LIN {X 0,Y 523.894,Z 140.721,A -85,B 0,C 180,E1 -4799.759,E2 -4799.759} C_VEL
LIN {X 0,Y 523.931,Z 140.719,A -85,B 0,C 180,E1 -4802.45,E2 -4802.45} C_VEL
LIN {X 0,Y 523.92,Z 140.722,A -85,B 0,C 180,E1 -4805.227,E2 -4805.227} C_VEL
LIN {X 0,Y 523.914,Z 140.72,A -85,B 0,C 180,E1 -4808.102,E2 -4808.102} C_VEL
LIN {X 0,Y 523.94,Z 140.717,A -85,B 0,C 180,E1 -4811.308,E2 -4811.308} C_VEL
LIN {X 0,Y 523.938,Z 140.723,A -85,B 0,C 180,E1 -4814.689,E2 -4814.689} C_VEL
LIN {X 0,Y 523.94,Z 140.717,A -85,B 0,C 180,E1 -4817.88,E2 -4817.88} C_VEL
LIN {X 0,Y 523.92,Z 140.72,A -85,B 0,C 180,E1 -4820.915,E2 -4820.915} C_VEL
LIN {X 0,Y 523.895,Z 140.724,A -85,B 0,C 180,E1 -4823.825,E2 -4823.825} C_VEL
LIN {X 0,Y 523.941,Z 140.719,A -85,B 0,C 180,E1 -4826.635,E2 -4826.635} C_VEL
LIN {X 0,Y 523.947,Z 140.715,A -85,B 0,C 180,E1 -4829.355,E2 -4829.355} C_VEL
LIN {X 0,Y 523.946,Z 140.721,A -85,B 0,C 180,E1 -4832.288,E2 -4832.288} C_VEL
LIN {X 0,Y 523.927,Z 140.719,A -85,B 0,C 180,E1 -4834.58,E2 -4834.58} C_VEL
LIN {X 0,Y 523.91,Z 140.72,A -85,B 0,C 180,E1 -4837.106,E2 -4837.106} C_VEL
LIN {X 0,Y 523.978,Z 140.72,A -85,B 0,C 180,E1 -4839.866,E2 -4839.866} C_VEL
LIN {X 0,Y 523.953,Z 140.714,A -85,B 0,C 180,E1 -4842.837,E2 -4842.837} C_VEL
LIN {X 0,Y 523.977,Z 140.714,A -85,B 0,C 180,E1 -4845.236,E2 -4845.236} C_VEL
LIN {X 0,Y 524.012,Z 140.707,A -85,B 0,C 180,E1 -4848.394,E2 -4848.394} C_VEL
LIN {X 0,Y 524,Z 140.717,A -85,B 0,C 180,E1 -4851.516,E2 -4851.516} C_VEL
LIN {X 0,Y 524.082,Z 140.699,A -85,B 0,C 180,E1 -4854.614,E2 -4854.614} C_VEL
LIN {X 0,Y 524.113,Z 140.698,A -85,B 0,C 180,E1 -4857.695,E2 -4857.695} C_VEL
LIN {X 0,Y 524.121,Z 140.696,A -85,B 0,C 180,E1 -4860.768,E2 -4860.768} C_VEL
LIN {X 0,Y 524.071,Z 140.708,A -85,B 0,C 180,E1 -4863.075,E2 -4863.075} C_VEL
LIN {X 0,Y 524.034,Z 140.704,A -85,B 0,C 180,E1 -4866.159,E2 -4866.159} C_VEL
LIN {X 0,Y 524.001,Z 140.711,A -85,B 0,C 180,E1 -4868.484,E2 -4868.484} C_VEL
LIN {X 0,Y 524.003,Z 140.708,A -85,B 0,C 180,E1 -4871.74,E2 -4871.74} C_VEL
LIN {X 0,Y 523.993,Z 140.714,A -85,B 0,C 180,E1 -4875.052,E2 -4875.052} C_VEL
LIN {X 0,Y 523.964,Z 140.713,A -85,B 0,C 180,E1 -4877.969,E2 -4877.969} C_VEL
LIN {X 0,Y 523.972,Z 140.717,A -85,B 0,C 180,E1 -4880.41,E2 -4880.41} C_VEL
LIN {X 0,Y 523.911,Z 140.723,A -85,B 0,C 180,E1 -4882.894,E2 -4882.894} C_VEL
LIN {X 0,Y 523.953,Z 140.714,A -85,B 0,C 180,E1 -4885.419,E2 -4885.419} C_VEL
LIN {X 0,Y 523.968,Z 140.716,A -85,B 0,C 180,E1 -4887.999,E2 -4887.999} C_VEL
LIN {X 0,Y 523.945,Z 140.717,A -85,B 0,C 180,E1 -4890.855,E2 -4890.855} C_VEL
LIN {X 0,Y 523.96,Z 140.716,A -85,B 0,C 180,E1 -4893.735,E2 -4893.735} C_VEL
LIN {X 0,Y 523.904,Z 140.725,A -85,B 0,C 180,E1 -4896.402,E2 -4896.402} C_VEL
LIN {X 0,Y 523.924,Z 140.718,A -85,B 0,C 180,E1 -4899.085,E2 -4899.085} C_VEL
LIN {X 0,Y 523.957,Z 140.72,A -85,B 0,C 180,E1 -4902.119,E2 -4902.119} C_VEL
LIN {X 0,Y 523.957,Z 140.715,A -85,B 0,C 180,E1 -4905.309,E2 -4905.309} C_VEL
LIN {X 0,Y 523.921,Z 140.718,A -85,B 0,C 180,E1 -4906.898,E2 -4906.898} C_VEL
LIN {X 0,Y 523.254,Z 140.808,A -85,B 0,C 180,E1 -4907.54,E2 -4907.54} C_VEL
LIN {X 0,Y 520.412,Z 141.161,A -85,B 0,C 180,E1 -4908.581,E2 -4908.581} C_VEL
LIN {X 0,Y 518.008,Z 141.461,A -85,B 0,C 180,E1 -4909.42,E2 -4909.42} C_VEL
LIN {X 0,Y 516.971,Z 141.589,A -85,B 0,C 180,E1 -4910.068,E2 -4910.068} C_VEL
LIN {X 0,Y 516.883,Z 141.597,A -85,B 0,C 180,E1 -4910.287,E2 -4910.287} C_VEL
LIN {X 0,Y 516.879,Z 141.6,A -85,B 0,C 180,E1 -4913.343,E2 -4913.343} C_VEL
LIN {X 0,Y 516.886,Z 141.596,A -85,B 0,C 180,E1 -4916.119,E2 -4916.119} C_VEL
LIN {X 0,Y 516.892,Z 141.596,A -85,B 0,C 180,E1 -4918.936,E2 -4918.936} C_VEL
LIN {X 0,Y 516.918,Z 141.598,A -85,B 0,C 180,E1 -4921.585,E2 -4921.585} C_VEL
LIN {X 0,Y 516.934,Z 141.59,A -85,B 0,C 180,E1 -4924.211,E2 -4924.211} C_VEL
LIN {X 0,Y 516.867,Z 141.601,A -85,B 0,C 180,E1 -4926.776,E2 -4926.776} C_VEL
LIN {X 0,Y 516.972,Z 141.775,A -85,B 0,C 180,E1 -4929.041,E2 -4929.041} C_VEL
LIN {X 0,Y 517.715,Z 147.463,A -85,B 0,C 180,E1 -4930.161,E2 -4930.161} C_VEL
LIN {X 0,Y 517.441,Z 161.62,A -85,B 0,C 180,E1 -4932.818,E2 -4932.818} C_VEL
LIN {X 0,Y 517.249,Z 171.826,A -85,B 0,C 180,E1 -4934.685,E2 -4934.685} C_VEL
LIN {X 0,Y 519.153,Z 182.577,A -85,B 0,C 180,E1 -4934.898,E2 -4934.898} C_VEL
LIN {X 0,Y 518.664,Z 279.186,A -85,B 0,C 180,E1 -4936.258,E2 -4936.258} C_VEL
LIN {X 0,Y 518.488,Z 292.359,A -85,B 0,C 180,E1 -4936.603,E2 -4936.603} C_VEL
LIN {X 0,Y 518.232,Z 304.457,A -85,B 0,C 180,E1 -4937.07,E2 -4937.07} C_VEL
LIN {X 0,Y 518.017,Z 315.553,A -85,B 0,C 180,E1 -4937.644,E2 -4937.644} C_VEL
LIN {X 0,Y 517.72,Z 326.26,A -85,B 0,C 180,E1 -4938.35,E2 -4938.35} C_VEL
LIN {X 0,Y 517.414,Z 336.963,A -85,B 0,C 180,E1 -4939.236,E2 -4939.236} C_VEL
LIN {X 0,Y 517.104,Z 346.594,A -85,B 0,C 180,E1 -4940.219,E2 -4940.219} C_VEL
LIN {X 0,Y 516.877,Z 354.481,A -85,B 0,C 180,E1 -4941.201,E2 -4941.201} C_VEL
LIN {X 0,Y 516.638,Z 362.196,A -85,B 0,C 180,E1 -4942.378,E2 -4942.378} C_VEL
LIN {X 0,Y 516.501,Z 369.27,A -85,B 0,C 180,E1 -4943.751,E2 -4943.751} C_VEL
LIN {X 0,Y 516.316,Z 373.987,A -85,B 0,C 180,E1 -4944.924,E2 -4944.924} C_VEL
LIN {X 0,Y 516.375,Z 377.597,A -85,B 0,C 180,E1 -4946.098,E2 -4946.098} C_VEL
LIN {X 0,Y 516.327,Z 379.464,A -85,B 0,C 180,E1 -4946.879,E2 -4946.879} C_VEL
LIN {X 0,Y 516.266,Z 380.874,A -85,B 0,C 180,E1 -4947.659,E2 -4947.659} C_VEL
LIN {X 0,Y 516.163,Z 382.495,A -85,B 0,C 180,E1 -4949.22,E2 -4949.22} C_VEL
LIN {X 0,Y 516.158,Z 382.733,A -85,B 0,C 180,E1 -4950,E2 -4950} C_VEL
LIN {X 0,Y 516.163,Z 382.55,A -85,B 0,C 180,E1 -4950.78,E2 -4950.78} C_VEL
LIN {X 0,Y 516.266,Z 381,A -85,B 0,C 180,E1 -4952.341,E2 -4952.341} C_VEL
LIN {X 0,Y 516.327,Z 379.645,A -85,B 0,C 180,E1 -4953.121,E2 -4953.121} C_VEL
LIN {X 0,Y 516.368,Z 376.78,A -85,B 0,C 180,E1 -4954.293,E2 -4954.293} C_VEL
LIN {X 0,Y 516.408,Z 372.896,A -85,B 0,C 180,E1 -4955.467,E2 -4955.467} C_VEL
LIN {X 0,Y 516.504,Z 366.966,A -85,B 0,C 180,E1 -4956.828,E2 -4956.828} C_VEL
LIN {X 0,Y 516.681,Z 360.354,A -85,B 0,C 180,E1 -4958.014,E2 -4958.014} C_VEL
LIN {X 0,Y 516.904,Z 352.199,A -85,B 0,C 180,E1 -4959.193,E2 -4959.193} C_VEL
LIN {X 0,Y 517.155,Z 343.853,A -85,B 0,C 180,E1 -4960.176,E2 -4960.176} C_VEL
LIN {X 0,Y 517.485,Z 333.549,A -85,B 0,C 180,E1 -4961.159,E2 -4961.159} C_VEL
LIN {X 0,Y 517.828,Z 322.274,A -85,B 0,C 180,E1 -4962.02,E2 -4962.02} C_VEL
LIN {X 0,Y 518.131,Z 310.364,A -85,B 0,C 180,E1 -4962.733,E2 -4962.733} C_VEL
LIN {X 0,Y 518.385,Z 298.344,A -85,B 0,C 180,E1 -4963.275,E2 -4963.275} C_VEL
LIN {X 0,Y 518.593,Z 285.267,A -85,B 0,C 180,E1 -4963.694,E2 -4963.694} C_VEL
LIN {X 0,Y 518.78,Z 272.765,A -85,B 0,C 180,E1 -4963.939,E2 -4963.939} C_VEL
LIN {X 0,Y 519.06,Z 182.069,A -85,B 0,C 180,E1 -4965.202,E2 -4965.202} C_VEL
LIN {X 0,Y 517.238,Z 171.844,A -85,B 0,C 180,E1 -4965.403,E2 -4965.403} C_VEL
LIN {X 0,Y 517.612,Z 155.547,A -85,B 0,C 180,E1 -4968.402,E2 -4968.402} C_VEL
LIN {X 0,Y 517.682,Z 146.406,A -85,B 0,C 180,E1 -4970.132,E2 -4970.132} C_VEL
LIN {X 0,Y 516.95,Z 141.595,A -85,B 0,C 180,E1 -4971.117,E2 -4971.117} C_VEL
LIN {X 0,Y 516.898,Z 141.598,A -85,B 0,C 180,E1 -4974.36,E2 -4974.36} C_VEL
LIN {X 0,Y 516.926,Z 141.598,A -85,B 0,C 180,E1 -4976.658,E2 -4976.658} C_VEL
LIN {X 0,Y 516.911,Z 141.592,A -85,B 0,C 180,E1 -4979.523,E2 -4979.523} C_VEL
LIN {X 0,Y 516.896,Z 141.602,A -85,B 0,C 180,E1 -4982.543,E2 -4982.543} C_VEL
LIN {X 0,Y 516.867,Z 141.597,A -85,B 0,C 180,E1 -4985.329,E2 -4985.329} C_VEL
LIN {X 0,Y 516.882,Z 141.598,A -85,B 0,C 180,E1 -4987.943,E2 -4987.943} C_VEL
LIN {X 0,Y 516.884,Z 141.598,A -85,B 0,C 180,E1 -4990.741,E2 -4990.741} C_VEL
LIN {X 0,Y 516.885,Z 141.596,A -85,B 0,C 180,E1 -4992.831,E2 -4992.831} C_VEL
LIN {X 0,Y 516.924,Z 141.59,A -85,B 0,C 180,E1 -4995.01,E2 -4995.01} C_VEL
LIN {X 0,Y 516.915,Z 141.595,A -85,B 0,C 180,E1 -4998.398,E2 -4998.398} C_VEL
LIN {X 0,Y 516.883,Z 141.596,A -85,B 0,C 180,E1 -5001.284,E2 -5001.284} C_VEL
LIN {X 0,Y 516.871,Z 141.601,A -85,B 0,C 180,E1 -5004.219,E2 -5004.219} C_VEL
LIN {X 0,Y 516.895,Z 141.594,A -85,B 0,C 180,E1 -5007.053,E2 -5007.053} C_VEL
LIN {X 0,Y 516.892,Z 141.602,A -85,B 0,C 180,E1 -5009.796,E2 -5009.796} C_VEL
LIN {X 0,Y 516.926,Z 141.59,A -85,B 0,C 180,E1 -5012.467,E2 -5012.467} C_VEL
LIN {X 0,Y 516.909,Z 141.594,A -85,B 0,C 180,E1 -5015.072,E2 -5015.072} C_VEL
LIN {X 0,Y 516.885,Z 141.595,A -85,B 0,C 180,E1 -5018.462,E2 -5018.462} C_VEL
LIN {X 0,Y 516.903,Z 141.595,A -85,B 0,C 180,E1 -5020.955,E2 -5020.955} C_VEL
LIN {X 0,Y 516.913,Z 141.599,A -85,B 0,C 180,E1 -5023.41,E2 -5023.41} C_VEL
LIN {X 0,Y 516.894,Z 141.595,A -85,B 0,C 180,E1 -5025.834,E2 -5025.834} C_VEL
LIN {X 0,Y 516.965,Z 141.585,A -85,B 0,C 180,E1 -5028.234,E2 -5028.234} C_VEL
LIN {X 0,Y 516.968,Z 141.589,A -85,B 0,C 180,E1 -5031.4,E2 -5031.4} C_VEL
LIN {X 0,Y 517.002,Z 141.581,A -85,B 0,C 180,E1 -5033.757,E2 -5033.757} C_VEL
LIN {X 0,Y 517.012,Z 141.588,A -85,B 0,C 180,E1 -5036.883,E2 -5036.883} C_VEL
LIN {X 0,Y 517.085,Z 141.57,A -85,B 0,C 180,E1 -5040,E2 -5040} C_VEL
LIN {X 0,Y 517.01,Z 141.582,A -85,B 0,C 180,E1 -5043.117,E2 -5043.117} C_VEL
LIN {X 0,Y 517.002,Z 141.584,A -85,B 0,C 180,E1 -5046.243,E2 -5046.243} C_VEL
LIN {X 0,Y 516.944,Z 141.587,A -85,B 0,C 180,E1 -5049.389,E2 -5049.389} C_VEL
LIN {X 0,Y 516.951,Z 141.587,A -85,B 0,C 180,E1 -5051.807,E2 -5051.807} C_VEL
LIN {X 0,Y 516.944,Z 141.588,A -85,B 0,C 180,E1 -5055.147,E2 -5055.147} C_VEL
LIN {X 0,Y 516.915,Z 141.599,A -85,B 0,C 180,E1 -5058.223,E2 -5058.223} C_VEL
LIN {X 0,Y 516.911,Z 141.593,A -85,B 0,C 180,E1 -5060.702,E2 -5060.702} C_VEL
LIN {X 0,Y 516.889,Z 141.603,A -85,B 0,C 180,E1 -5064.073,E2 -5064.073} C_VEL
LIN {X 0,Y 516.92,Z 141.591,A -85,B 0,C 180,E1 -5066.658,E2 -5066.658} C_VEL
LIN {X 0,Y 516.909,Z 141.595,A -85,B 0,C 180,E1 -5069.524,E2 -5069.524} C_VEL
LIN {X 0,Y 516.895,Z 141.594,A -85,B 0,C 180,E1 -5072.543,E2 -5072.543} C_VEL
LIN {X 0,Y 516.863,Z 141.601,A -85,B 0,C 180,E1 -5075.329,E2 -5075.329} C_VEL
LIN {X 0,Y 516.878,Z 141.6,A -85,B 0,C 180,E1 -5077.943,E2 -5077.943} C_VEL
LIN {X 0,Y 516.88,Z 141.595,A -85,B 0,C 180,E1 -5080.742,E2 -5080.742} C_VEL
LIN {X 0,Y 516.881,Z 141.598,A -85,B 0,C 180,E1 -5083.904,E2 -5083.904} C_VEL
LIN {X 0,Y 516.88,Z 141.596,A -85,B 0,C 180,E1 -5086.107,E2 -5086.107} C_VEL
LIN {X 0,Y 516.902,Z 141.593,A -85,B 0,C 180,E1 -5088.4,E2 -5088.4} C_VEL
LIN {X 0,Y 516.877,Z 141.604,A -85,B 0,C 180,E1 -5091.284,E2 -5091.284} C_VEL
LIN {X 0,Y 516.871,Z 141.596,A -85,B 0,C 180,E1 -5094.22,E2 -5094.22} C_VEL
LIN {X 0,Y 516.88,Z 141.604,A -85,B 0,C 180,E1 -5097.052,E2 -5097.052} C_VEL
LIN {X 0,Y 516.863,Z 141.6,A -85,B 0,C 180,E1 -5099.795,E2 -5099.795} C_VEL
LIN {X 0,Y 516.877,Z 141.599,A -85,B 0,C 180,E1 -5102.465,E2 -5102.465} C_VEL
LIN {X 0,Y 516.846,Z 141.608,A -85,B 0,C 180,E1 -5105.069,E2 -5105.069} C_VEL
LIN {X 0,Y 516.902,Z 141.692,A -85,B 0,C 180,E1 -5105.981,E2 -5105.981} C_VEL
LIN {X 0,Y 518.288,Z 149.569,A -85,B 0,C 180,E1 -5107.372,E2 -5107.372} C_VEL
LIN {X 0,Y 517.935,Z 164.192,A -85,B 0,C 180,E1 -5109.793,E2 -5109.793} C_VEL
LIN {X 0,Y 517.529,Z 180.375,A -85,B 0,C 180,E1 -5112.437,E2 -5112.437} C_VEL
LIN {X 0,Y 517.238,Z 194.025,A -85,B 0,C 180,E1 -5114.635,E2 -5114.635} C_VEL
LIN {X 0,Y 519.105,Z 206.824,A -85,B 0,C 180,E1 -5114.871,E2 -5114.871} C_VEL
LIN {X 0,Y 518.632,Z 301.977,A -85,B 0,C 180,E1 -5116.207,E2 -5116.207} C_VEL
LIN {X 0,Y 518.385,Z 315.258,A -85,B 0,C 180,E1 -5116.55,E2 -5116.55} C_VEL
LIN {X 0,Y 518.1,Z 328.548,A -85,B 0,C 180,E1 -5117.067,E2 -5117.067} C_VEL
LIN {X 0,Y 517.775,Z 340.338,A -85,B 0,C 180,E1 -5117.696,E2 -5117.696} C_VEL
LIN {X 0,Y 517.491,Z 352.593,A -85,B 0,C 180,E1 -5118.544,E2 -5118.544} C_VEL
LIN {X 0,Y 517.171,Z 362.784,A -85,B 0,C 180,E1 -5119.429,E2 -5119.429} C_VEL
LIN {X 0,Y 516.926,Z 371.954,A -85,B 0,C 180,E1 -5120.413,E2 -5120.413} C_VEL
LIN {X 0,Y 516.653,Z 380.888,A -85,B 0,C 180,E1 -5121.591,E2 -5121.591} C_VEL
LIN {X 0,Y 516.503,Z 388.079,A -85,B 0,C 180,E1 -5122.769,E2 -5122.769} C_VEL
LIN {X 0,Y 516.407,Z 394.627,A -85,B 0,C 180,E1 -5124.142,E2 -5124.142} C_VEL
LIN {X 0,Y 516.267,Z 398.957,A -85,B 0,C 180,E1 -5125.315,E2 -5125.315} C_VEL
LIN {X 0,Y 516.352,Z 401.252,A -85,B 0,C 180,E1 -5126.098,E2 -5126.098} C_VEL
LIN {X 0,Y 516.282,Z 403.109,A -85,B 0,C 180,E1 -5126.879,E2 -5126.879} C_VEL
LIN {X 0,Y 516.261,Z 404.502,A -85,B 0,C 180,E1 -5127.659,E2 -5127.659} C_VEL
LIN {X 0,Y 516.161,Z 406.101,A -85,B 0,C 180,E1 -5129.22,E2 -5129.22} C_VEL
LIN {X 0,Y 516.157,Z 406.317,A -85,B 0,C 180,E1 -5130,E2 -5130} C_VEL
LIN {X 0,Y 516.192,Z 405.496,A -85,B 0,C 180,E1 -5131.56,E2 -5131.56} C_VEL
LIN {X 0,Y 516.261,Z 404.505,A -85,B 0,C 180,E1 -5132.341,E2 -5132.341} C_VEL
LIN {X 0,Y 516.282,Z 403.112,A -85,B 0,C 180,E1 -5133.121,E2 -5133.121} C_VEL
LIN {X 0,Y 516.31,Z 400.182,A -85,B 0,C 180,E1 -5134.294,E2 -5134.294} C_VEL
LIN {X 0,Y 516.39,Z 396.216,A -85,B 0,C 180,E1 -5135.467,E2 -5135.467} C_VEL
LIN {X 0,Y 516.442,Z 390.346,A -85,B 0,C 180,E1 -5136.794,E2 -5136.794} C_VEL
LIN {X 0,Y 516.587,Z 383.445,A -85,B 0,C 180,E1 -5138.016,E2 -5138.016} C_VEL
LIN {X 0,Y 516.806,Z 375.171,A -85,B 0,C 180,E1 -5139.195,E2 -5139.195} C_VEL
LIN {X 0,Y 517.021,Z 366.689,A -85,B 0,C 180,E1 -5140.178,E2 -5140.178} C_VEL
LIN {X 0,Y 517.372,Z 356.209,A -85,B 0,C 180,E1 -5141.161,E2 -5141.161} C_VEL
LIN {X 0,Y 517.674,Z 345.063,A -85,B 0,C 180,E1 -5142.003,E2 -5142.003} C_VEL
LIN {X 0,Y 517.96,Z 334.472,A -85,B 0,C 180,E1 -5142.638,E2 -5142.638} C_VEL
LIN {X 0,Y 518.236,Z 322.813,A -85,B 0,C 180,E1 -5143.179,E2 -5143.179} C_VEL
LIN {X 0,Y 518.494,Z 309.377,A -85,B 0,C 180,E1 -5143.622,E2 -5143.622} C_VEL
LIN {X 0,Y 518.708,Z 296.109,A -85,B 0,C 180,E1 -5143.891,E2 -5143.891} C_VEL
LIN {X 0,Y 518.988,Z 204.886,A -85,B 0,C 180,E1 -5145.16,E2 -5145.16} C_VEL
LIN {X 0,Y 517.226,Z 193.828,A -85,B 0,C 180,E1 -5145.388,E2 -5145.388} C_VEL
LIN {X 0,Y 517.68,Z 175.231,A -85,B 0,C 180,E1 -5148.399,E2 -5148.399} C_VEL
LIN {X 0,Y 518.165,Z 157.709,A -85,B 0,C 180,E1 -5151.273,E2 -5151.273} C_VEL
LIN {X 0,Y 518.259,Z 148.792,A -85,B 0,C 180,E1 -5152.759,E2 -5152.759} C_VEL
LIN {X 0,Y 516.887,Z 141.601,A -85,B 0,C 180,E1 -5154.073,E2 -5154.073} C_VEL
LIN {X 0,Y 516.85,Z 141.604,A -85,B 0,C 180,E1 -5156.662,E2 -5156.662} C_VEL
LIN {X 0,Y 516.886,Z 141.596,A -85,B 0,C 180,E1 -5159.518,E2 -5159.518} C_VEL
LIN {X 0,Y 516.892,Z 141.597,A -85,B 0,C 180,E1 -5162.542,E2 -5162.542} C_VEL
LIN {X 0,Y 516.866,Z 141.6,A -85,B 0,C 180,E1 -5165.329,E2 -5165.329} C_VEL
LIN {X 0,Y 516.879,Z 141.596,A -85,B 0,C 180,E1 -5167.943,E2 -5167.943} C_VEL
LIN {X 0,Y 516.864,Z 141.606,A -85,B 0,C 180,E1 -5170.743,E2 -5170.743} C_VEL
LIN {X 0,Y 516.854,Z 141.604,A -85,B 0,C 180,E1 -5172.834,E2 -5172.834} C_VEL
LIN {X 0,Y 516.895,Z 141.596,A -85,B 0,C 180,E1 -5175.007,E2 -5175.007} C_VEL
LIN {X 0,Y 516.908,Z 141.6,A -85,B 0,C 180,E1 -5178.399,E2 -5178.399} C_VEL
LIN {X 0,Y 516.88,Z 141.595,A -85,B 0,C 180,E1 -5181.284,E2 -5181.284} C_VEL
LIN {X 0,Y 516.867,Z 141.605,A -85,B 0,C 180,E1 -5184.219,E2 -5184.219} C_VEL
LIN {X 0,Y 516.894,Z 141.594,A -85,B 0,C 180,E1 -5187.053,E2 -5187.053} C_VEL
LIN {X 0,Y 516.885,Z 141.599,A -85,B 0,C 180,E1 -5189.796,E2 -5189.796} C_VEL
LIN {X 0,Y 516.898,Z 141.596,A -85,B 0,C 180,E1 -5192.466,E2 -5192.466} C_VEL
LIN {X 0,Y 516.865,Z 141.597,A -85,B 0,C 180,E1 -5195.069,E2 -5195.069} C_VEL
LIN {X 0,Y 516.868,Z 141.602,A -85,B 0,C 180,E1 -5197.621,E2 -5197.621} C_VEL
LIN {X 0,Y 516.931,Z 141.593,A -85,B 0,C 180,E1 -5200.13,E2 -5200.13} C_VEL
LIN {X 0,Y 516.905,Z 141.592,A -85,B 0,C 180,E1 -5202.595,E2 -5202.595} C_VEL
LIN {X 0,Y 516.942,Z 141.589,A -85,B 0,C 180,E1 -5205.03,E2 -5205.03} C_VEL
LIN {X 0,Y 516.965,Z 141.586,A -85,B 0,C 180,E1 -5208.234,E2 -5208.234} C_VEL
LIN {X 0,Y 516.965,Z 141.592,A -85,B 0,C 180,E1 -5211.4,E2 -5211.4} C_VEL
LIN {X 0,Y 517.002,Z 141.584,A -85,B 0,C 180,E1 -5213.757,E2 -5213.757} C_VEL
LIN {X 0,Y 517.01,Z 141.582,A -85,B 0,C 180,E1 -5216.883,E2 -5216.883} C_VEL
LIN {X 0,Y 517.085,Z 141.57,A -85,B 0,C 180,E1 -5220,E2 -5220} C_VEL
LIN {X 0,Y 517.012,Z 141.588,A -85,B 0,C 180,E1 -5223.117,E2 -5223.117} C_VEL
LIN {X 0,Y 516.995,Z 141.581,A -85,B 0,C 180,E1 -5226.243,E2 -5226.243} C_VEL
LIN {X 0,Y 516.965,Z 141.588,A -85,B 0,C 180,E1 -5228.6,E2 -5228.6} C_VEL
LIN {X 0,Y 516.952,Z 141.586,A -85,B 0,C 180,E1 -5231.807,E2 -5231.807} C_VEL
LIN {X 0,Y 516.944,Z 141.591,A -85,B 0,C 180,E1 -5235.147,E2 -5235.147} C_VEL
LIN {X 0,Y 516.925,Z 141.592,A -85,B 0,C 180,E1 -5238.222,E2 -5238.222} C_VEL
LIN {X 0,Y 516.913,Z 141.599,A -85,B 0,C 180,E1 -5240.702,E2 -5240.702} C_VEL
LIN {X 0,Y 516.904,Z 141.595,A -85,B 0,C 180,E1 -5244.073,E2 -5244.073} C_VEL
LIN {X 0,Y 516.925,Z 141.595,A -85,B 0,C 180,E1 -5246.658,E2 -5246.658} C_VEL
LIN {X 0,Y 516.911,Z 141.592,A -85,B 0,C 180,E1 -5249.524,E2 -5249.524} C_VEL
LIN {X 0,Y 516.896,Z 141.598,A -85,B 0,C 180,E1 -5252.544,E2 -5252.544} C_VEL
LIN {X 0,Y 516.867,Z 141.597,A -85,B 0,C 180,E1 -5255.33,E2 -5255.33} C_VEL
LIN {X 0,Y 516.882,Z 141.602,A -85,B 0,C 180,E1 -5257.943,E2 -5257.943} C_VEL
LIN {X 0,Y 516.886,Z 141.595,A -85,B 0,C 180,E1 -5260.742,E2 -5260.742} C_VEL
LIN {X 0,Y 516.885,Z 141.595,A -85,B 0,C 180,E1 -5262.831,E2 -5262.831} C_VEL
LIN {X 0,Y 516.924,Z 141.59,A -85,B 0,C 180,E1 -5265.01,E2 -5265.01} C_VEL
LIN {X 0,Y 516.917,Z 141.592,A -85,B 0,C 180,E1 -5268.399,E2 -5268.399} C_VEL
LIN {X 0,Y 516.883,Z 141.597,A -85,B 0,C 180,E1 -5270.287,E2 -5270.287} C_VEL
LIN {X 0,Y 516.211,Z 141.679,A -85,B 0,C 180,E1 -5270.937,E2 -5270.937} C_VEL
LIN {X 0,Y 513.365,Z 142.042,A -85,B 0,C 180,E1 -5271.993,E2 -5271.993} C_VEL
LIN {X 0,Y 510.957,Z 142.347,A -85,B 0,C 180,E1 -5272.843,E2 -5272.843} C_VEL
LIN {X 0,Y 509.913,Z 142.474,A -85,B 0,C 180,E1 -5273.499,E2 -5273.499} C_VEL
LIN {X 0,Y 509.822,Z 142.482,A -85,B 0,C 180,E1 -5273.722,E2 -5273.722} C_VEL
LIN {X 0,Y 509.843,Z 142.472,A -85,B 0,C 180,E1 -5276.538,E2 -5276.538} C_VEL
LIN {X 0,Y 509.845,Z 142.479,A -85,B 0,C 180,E1 -5279.334,E2 -5279.334} C_VEL
LIN {X 0,Y 509.892,Z 142.467,A -85,B 0,C 180,E1 -5282.055,E2 -5282.055} C_VEL
LIN {X 0,Y 509.878,Z 142.471,A -85,B 0,C 180,E1 -5284.704,E2 -5284.704} C_VEL
LIN {X 0,Y 509.829,Z 142.48,A -85,B 0,C 180,E1 -5287.458,E2 -5287.458} C_VEL
LIN {X 0,Y 509.909,Z 142.617,A -85,B 0,C 180,E1 -5288.895,E2 -5288.895} C_VEL
LIN {X 0,Y 510.762,Z 148.591,A -85,B 0,C 180,E1 -5290.089,E2 -5290.089} C_VEL
LIN {X 0,Y 510.48,Z 161.707,A -85,B 0,C 180,E1 -5292.576,E2 -5292.576} C_VEL
LIN {X 0,Y 510.268,Z 171.957,A -85,B 0,C 180,E1 -5294.47,E2 -5294.47} C_VEL
LIN {X 0,Y 512.319,Z 183.37,A -85,B 0,C 180,E1 -5294.7,E2 -5294.7} C_VEL
LIN {X 0,Y 511.789,Z 279.376,A -85,B 0,C 180,E1 -5296.07,E2 -5296.07} C_VEL
LIN {X 0,Y 511.585,Z 292.541,A -85,B 0,C 180,E1 -5296.418,E2 -5296.418} C_VEL
LIN {X 0,Y 511.29,Z 305.746,A -85,B 0,C 180,E1 -5296.942,E2 -5296.942} C_VEL
LIN {X 0,Y 510.991,Z 318.287,A -85,B 0,C 180,E1 -5297.633,E2 -5297.633} C_VEL
LIN {X 0,Y 510.709,Z 329.005,A -85,B 0,C 180,E1 -5298.389,E2 -5298.389} C_VEL
LIN {X 0,Y 510.357,Z 339.261,A -85,B 0,C 180,E1 -5299.286,E2 -5299.286} C_VEL
LIN {X 0,Y 510.062,Z 348.463,A -85,B 0,C 180,E1 -5300.283,E2 -5300.283} C_VEL
LIN {X 0,Y 509.747,Z 357.393,A -85,B 0,C 180,E1 -5301.477,E2 -5301.477} C_VEL
LIN {X 0,Y 509.517,Z 364.584,A -85,B 0,C 180,E1 -5302.67,E2 -5302.67} C_VEL
LIN {X 0,Y 509.429,Z 369.435,A -85,B 0,C 180,E1 -5303.664,E2 -5303.664} C_VEL
LIN {X 0,Y 509.251,Z 374.152,A -85,B 0,C 180,E1 -5304.853,E2 -5304.853} C_VEL
LIN {X 0,Y 509.307,Z 377.76,A -85,B 0,C 180,E1 -5306.044,E2 -5306.044} C_VEL
LIN {X 0,Y 509.241,Z 379.628,A -85,B 0,C 180,E1 -5306.835,E2 -5306.835} C_VEL
LIN {X 0,Y 509.196,Z 381.037,A -85,B 0,C 180,E1 -5307.627,E2 -5307.627} C_VEL
LIN {X 0,Y 509.076,Z 382.658,A -85,B 0,C 180,E1 -5309.209,E2 -5309.209} C_VEL
LIN {X 0,Y 509.069,Z 382.895,A -85,B 0,C 180,E1 -5310,E2 -5310} C_VEL
LIN {X 0,Y 509.076,Z 382.711,A -85,B 0,C 180,E1 -5310.791,E2 -5310.791} C_VEL
LIN {X 0,Y 509.196,Z 381.161,A -85,B 0,C 180,E1 -5312.373,E2 -5312.373} C_VEL
LIN {X 0,Y 509.242,Z 379.806,A -85,B 0,C 180,E1 -5313.164,E2 -5313.164} C_VEL
LIN {X 0,Y 509.29,Z 376.941,A -85,B 0,C 180,E1 -5314.353,E2 -5314.353} C_VEL
LIN {X 0,Y 509.354,Z 373.056,A -85,B 0,C 180,E1 -5315.542,E2 -5315.542} C_VEL
LIN {X 0,Y 509.431,Z 367.355,A -85,B 0,C 180,E1 -5316.878,E2 -5316.878} C_VEL
LIN {X 0,Y 509.642,Z 360.512,A -85,B 0,C 180,E1 -5318.126,E2 -5318.126} C_VEL
LIN {X 0,Y 509.885,Z 352.357,A -85,B 0,C 180,E1 -5319.32,E2 -5319.32} C_VEL
LIN {X 0,Y 510.148,Z 344.01,A -85,B 0,C 180,E1 -5320.317,E2 -5320.317} C_VEL
LIN {X 0,Y 510.534,Z 333.704,A -85,B 0,C 180,E1 -5321.313,E2 -5321.313} C_VEL
LIN {X 0,Y 510.879,Z 322.134,A -85,B 0,C 180,E1 -5322.206,E2 -5322.206} C_VEL
LIN {X 0,Y 511.196,Z 310.514,A -85,B 0,C 180,E1 -5322.909,E2 -5322.909} C_VEL
LIN {X 0,Y 511.484,Z 298.49,A -85,B 0,C 180,E1 -5323.458,E2 -5323.458} C_VEL
LIN {X 0,Y 511.71,Z 285.406,A -85,B 0,C 180,E1 -5323.882,E2 -5323.882} C_VEL
LIN {X 0,Y 511.899,Z 272.883,A -85,B 0,C 180,E1 -5324.13,E2 -5324.13} C_VEL
LIN {X 0,Y 512.182,Z 182.621,A -85,B 0,C 180,E1 -5325.405,E2 -5325.405} C_VEL
LIN {X 0,Y 510.267,Z 171.897,A -85,B 0,C 180,E1 -5325.631,E2 -5325.631} C_VEL
LIN {X 0,Y 510.662,Z 154.515,A -85,B 0,C 180,E1 -5328.87,E2 -5328.87} C_VEL
LIN {X 0,Y 510.556,Z 146.331,A -85,B 0,C 180,E1 -5330.447,E2 -5330.447} C_VEL
LIN {X 0,Y 509.91,Z 142.472,A -85,B 0,C 180,E1 -5331.264,E2 -5331.264} C_VEL
LIN {X 0,Y 509.857,Z 142.476,A -85,B 0,C 180,E1 -5334.527,E2 -5334.527} C_VEL
LIN {X 0,Y 509.885,Z 142.471,A -85,B 0,C 180,E1 -5337.055,E2 -5337.055} C_VEL
LIN {X 0,Y 509.859,Z 142.47,A -85,B 0,C 180,E1 -5339.751,E2 -5339.751} C_VEL
LIN {X 0,Y 509.868,Z 142.474,A -85,B 0,C 180,E1 -5342.773,E2 -5342.773} C_VEL
LIN {X 0,Y 509.827,Z 142.474,A -85,B 0,C 180,E1 -5345.578,E2 -5345.578} C_VEL
LIN {X 0,Y 509.851,Z 142.479,A -85,B 0,C 180,E1 -5348.338,E2 -5348.338} C_VEL
LIN {X 0,Y 509.856,Z 142.47,A -85,B 0,C 180,E1 -5351.425,E2 -5351.425} C_VEL
LIN {X 0,Y 509.858,Z 142.473,A -85,B 0,C 180,E1 -5354.668,E2 -5354.668} C_VEL
LIN {X 0,Y 509.858,Z 142.479,A -85,B 0,C 180,E1 -5358.103,E2 -5358.103} C_VEL
LIN {X 0,Y 509.848,Z 142.472,A -85,B 0,C 180,E1 -5360.647,E2 -5360.647} C_VEL
LIN {X 0,Y 509.825,Z 142.479,A -85,B 0,C 180,E1 -5363.647,E2 -5363.647} C_VEL
LIN {X 0,Y 509.859,Z 142.471,A -85,B 0,C 180,E1 -5366.539,E2 -5366.539} C_VEL
LIN {X 0,Y 509.845,Z 142.475,A -85,B 0,C 180,E1 -5369.334,E2 -5369.334} C_VEL
LIN {X 0,Y 509.892,Z 142.469,A -85,B 0,C 180,E1 -5372.054,E2 -5372.054} C_VEL
LIN {X 0,Y 509.876,Z 142.468,A -85,B 0,C 180,E1 -5374.704,E2 -5374.704} C_VEL
LIN {X 0,Y 509.826,Z 142.482,A -85,B 0,C 180,E1 -5377.458,E2 -5377.458} C_VEL
LIN {X 0,Y 509.917,Z 142.466,A -85,B 0,C 180,E1 -5379.845,E2 -5379.845} C_VEL
LIN {X 0,Y 509.884,Z 142.473,A -85,B 0,C 180,E1 -5383.175,E2 -5383.175} C_VEL
LIN {X 0,Y 509.863,Z 142.473,A -85,B 0,C 180,E1 -5385.634,E2 -5385.634} C_VEL
LIN {X 0,Y 509.913,Z 142.468,A -85,B 0,C 180,E1 -5388.874,E2 -5388.874} C_VEL
LIN {X 0,Y 509.951,Z 142.458,A -85,B 0,C 180,E1 -5392.078,E2 -5392.078} C_VEL
LIN {X 0,Y 509.979,Z 142.457,A -85,B 0,C 180,E1 -5394.464,E2 -5394.464} C_VEL
LIN {X 0,Y 510.055,Z 142.446,A -85,B 0,C 180,E1 -5397.631,E2 -5397.631} C_VEL
LIN {X 0,Y 510.064,Z 142.453,A -85,B 0,C 180,E1 -5400.789,E2 -5400.789} C_VEL
LIN {X 0,Y 509.952,Z 142.461,A -85,B 0,C 180,E1 -5403.16,E2 -5403.16} C_VEL
LIN {X 0,Y 509.953,Z 142.463,A -85,B 0,C 180,E1 -5406.33,E2 -5406.33} C_VEL
LIN {X 0,Y 509.91,Z 142.47,A -85,B 0,C 180,E1 -5408.72,E2 -5408.72} C_VEL
LIN {X 0,Y 509.904,Z 142.466,A -85,B 0,C 180,E1 -5411.932,E2 -5411.932} C_VEL
LIN {X 0,Y 509.893,Z 142.466,A -85,B 0,C 180,E1 -5415.242,E2 -5415.242} C_VEL
LIN {X 0,Y 509.86,Z 142.475,A -85,B 0,C 180,E1 -5418.484,E2 -5418.484} C_VEL
LIN {X 0,Y 509.849,Z 142.471,A -85,B 0,C 180,E1 -5421.002,E2 -5421.002} C_VEL
LIN {X 0,Y 509.821,Z 142.477,A -85,B 0,C 180,E1 -5423.564,E2 -5423.564} C_VEL
LIN {X 0,Y 509.908,Z 142.467,A -85,B 0,C 180,E1 -5426.378,E2 -5426.378} C_VEL
LIN {X 0,Y 509.871,Z 142.468,A -85,B 0,C 180,E1 -5428.845,E2 -5428.845} C_VEL
LIN {X 0,Y 509.819,Z 142.48,A -85,B 0,C 180,E1 -5431.59,E2 -5431.59} C_VEL
LIN {X 0,Y 509.846,Z 142.473,A -85,B 0,C 180,E1 -5434.414,E2 -5434.414} C_VEL
LIN {X 0,Y 509.808,Z 142.48,A -85,B 0,C 180,E1 -5437.342,E2 -5437.342} C_VEL
LIN {X 0,Y 509.837,Z 142.473,A -85,B 0,C 180,E1 -5440.383,E2 -5440.383} C_VEL
LIN {X 0,Y 509.804,Z 142.48,A -85,B 0,C 180,E1 -5443.06,E2 -5443.06} C_VEL
LIN {X 0,Y 509.821,Z 142.478,A -85,B 0,C 180,E1 -5445.794,E2 -5445.794} C_VEL
LIN {X 0,Y 509.844,Z 142.472,A -85,B 0,C 180,E1 -5448.574,E2 -5448.574} C_VEL
LIN {X 0,Y 509.85,Z 142.473,A -85,B 0,C 180,E1 -5451.787,E2 -5451.787} C_VEL
LIN {X 0,Y 509.829,Z 142.476,A -85,B 0,C 180,E1 -5454.622,E2 -5454.622} C_VEL
LIN {X 0,Y 509.858,Z 142.473,A -85,B 0,C 180,E1 -5457.481,E2 -5457.481} C_VEL
LIN {X 0,Y 509.853,Z 142.474,A -85,B 0,C 180,E1 -5460.275,E2 -5460.275} C_VEL
LIN {X 0,Y 509.828,Z 142.482,A -85,B 0,C 180,E1 -5462.941,E2 -5462.941} C_VEL
LIN {X 0,Y 509.867,Z 142.631,A -85,B 0,C 180,E1 -5465.818,E2 -5465.818} C_VEL
LIN {X 0,Y 511.34,Z 151.29,A -85,B 0,C 180,E1 -5467.366,E2 -5467.366} C_VEL
LIN {X 0,Y 510.972,Z 164.412,A -85,B 0,C 180,E1 -5469.568,E2 -5469.568} C_VEL
LIN {X 0,Y 510.526,Z 181.323,A -85,B 0,C 180,E1 -5472.371,E2 -5472.371} C_VEL
LIN {X 0,Y 510.232,Z 193.729,A -85,B 0,C 180,E1 -5474.406,E2 -5474.406} C_VEL
LIN {X 0,Y 512.219,Z 206.578,A -85,B 0,C 180,E1 -5474.661,E2 -5474.661} C_VEL
LIN {X 0,Y 511.738,Z 301.814,A -85,B 0,C 180,E1 -5476.018,E2 -5476.018} C_VEL
LIN {X 0,Y 511.497,Z 315.096,A -85,B 0,C 180,E1 -5476.366,E2 -5476.366} C_VEL
LIN {X 0,Y 511.225,Z 327.263,A -85,B 0,C 180,E1 -5476.839,E2 -5476.839} C_VEL
LIN {X 0,Y 510.891,Z 338.778,A -85,B 0,C 180,E1 -5477.44,E2 -5477.44} C_VEL
LIN {X 0,Y 510.597,Z 349.842,A -85,B 0,C 180,E1 -5478.186,E2 -5478.186} C_VEL
LIN {X 0,Y 510.264,Z 360.505,A -85,B 0,C 180,E1 -5479.083,E2 -5479.083} C_VEL
LIN {X 0,Y 509.922,Z 370.112,A -85,B 0,C 180,E1 -5480.08,E2 -5480.08} C_VEL
LIN {X 0,Y 509.667,Z 377.987,A -85,B 0,C 180,E1 -5481.076,E2 -5481.076} C_VEL
LIN {X 0,Y 509.469,Z 385.679,A -85,B 0,C 180,E1 -5482.27,E2 -5482.27} C_VEL
LIN {X 0,Y 509.308,Z 392.768,A -85,B 0,C 180,E1 -5483.662,E2 -5483.662} C_VEL
LIN {X 0,Y 509.245,Z 397.485,A -85,B 0,C 180,E1 -5484.853,E2 -5484.853} C_VEL
LIN {X 0,Y 509.245,Z 401.089,A -85,B 0,C 180,E1 -5486.043,E2 -5486.043} C_VEL
LIN {X 0,Y 509.2,Z 402.947,A -85,B 0,C 180,E1 -5486.835,E2 -5486.835} C_VEL
LIN {X 0,Y 509.19,Z 404.34,A -85,B 0,C 180,E1 -5487.627,E2 -5487.627} C_VEL
LIN {X 0,Y 509.075,Z 405.939,A -85,B 0,C 180,E1 -5489.209,E2 -5489.209} C_VEL
LIN {X 0,Y 509.068,Z 406.155,A -85,B 0,C 180,E1 -5490,E2 -5490} C_VEL
LIN {X 0,Y 509.112,Z 405.335,A -85,B 0,C 180,E1 -5491.582,E2 -5491.582} C_VEL
LIN {X 0,Y 509.19,Z 404.343,A -85,B 0,C 180,E1 -5492.373,E2 -5492.373} C_VEL
LIN {X 0,Y 509.2,Z 402.95,A -85,B 0,C 180,E1 -5493.165,E2 -5493.165} C_VEL
LIN {X 0,Y 509.203,Z 400.02,A -85,B 0,C 180,E1 -5494.354,E2 -5494.354} C_VEL
LIN {X 0,Y 509.301,Z 396.054,A -85,B 0,C 180,E1 -5495.543,E2 -5495.543} C_VEL
LIN {X 0,Y 509.369,Z 390.405,A -85,B 0,C 180,E1 -5496.845,E2 -5496.845} C_VEL
LIN {X 0,Y 509.537,Z 383.283,A -85,B 0,C 180,E1 -5498.128,E2 -5498.128} C_VEL
LIN {X 0,Y 509.753,Z 375.008,A -85,B 0,C 180,E1 -5499.323,E2 -5499.323} C_VEL
LIN {X 0,Y 510.004,Z 366.526,A -85,B 0,C 180,E1 -5500.32,E2 -5500.32} C_VEL
LIN {X 0,Y 510.379,Z 356.046,A -85,B 0,C 180,E1 -5501.316,E2 -5501.316} C_VEL
LIN {X 0,Y 510.691,Z 345.756,A -85,B 0,C 180,E1 -5502.109,E2 -5502.109} C_VEL
LIN {X 0,Y 511.025,Z 334.309,A -85,B 0,C 180,E1 -5502.813,E2 -5502.813} C_VEL
LIN {X 0,Y 511.342,Z 322.651,A -85,B 0,C 180,E1 -5503.36,E2 -5503.36} C_VEL
LIN {X 0,Y 511.587,Z 310.13,A -85,B 0,C 180,E1 -5503.784,E2 -5503.784} C_VEL
LIN {X 0,Y 511.817,Z 297.462,A -85,B 0,C 180,E1 -5504.056,E2 -5504.056} C_VEL
LIN {X 0,Y 512.168,Z 205.96,A -85,B 0,C 180,E1 -5505.349,E2 -5505.349} C_VEL
LIN {X 0,Y 510.224,Z 193.76,A -85,B 0,C 180,E1 -5505.589,E2 -5505.589} C_VEL
LIN {X 0,Y 510.722,Z 175.072,A -85,B 0,C 180,E1 -5508.659,E2 -5508.659} C_VEL
LIN {X 0,Y 511.196,Z 157.55,A -85,B 0,C 180,E1 -5511.578,E2 -5511.578} C_VEL
LIN {X 0,Y 511.255,Z 149.602,A -85,B 0,C 180,E1 -5512.924,E2 -5512.924} C_VEL
LIN {X 0,Y 509.861,Z 142.476,A -85,B 0,C 180,E1 -5514.21,E2 -5514.21} C_VEL
LIN {X 0,Y 509.828,Z 142.48,A -85,B 0,C 180,E1 -5517.059,E2 -5517.059} C_VEL
LIN {X 0,Y 509.852,Z 142.47,A -85,B 0,C 180,E1 -5519.751,E2 -5519.751} C_VEL
LIN {X 0,Y 509.844,Z 142.478,A -85,B 0,C 180,E1 -5522.769,E2 -5522.769} C_VEL
LIN {X 0,Y 509.826,Z 142.475,A -85,B 0,C 180,E1 -5525.578,E2 -5525.578} C_VEL
LIN {X 0,Y 509.848,Z 142.474,A -85,B 0,C 180,E1 -5528.338,E2 -5528.338} C_VEL
LIN {X 0,Y 509.844,Z 142.472,A -85,B 0,C 180,E1 -5531.427,E2 -5531.427} C_VEL
LIN {X 0,Y 509.839,Z 142.48,A -85,B 0,C 180,E1 -5534.67,E2 -5534.67} C_VEL
LIN {X 0,Y 509.848,Z 142.475,A -85,B 0,C 180,E1 -5538.104,E2 -5538.104} C_VEL
LIN {X 0,Y 509.846,Z 142.477,A -85,B 0,C 180,E1 -5540.647,E2 -5540.647} C_VEL
LIN {X 0,Y 509.809,Z 142.477,A -85,B 0,C 180,E1 -5543.645,E2 -5543.645} C_VEL
LIN {X 0,Y 509.858,Z 142.474,A -85,B 0,C 180,E1 -5546.539,E2 -5546.539} C_VEL
LIN {X 0,Y 509.841,Z 142.472,A -85,B 0,C 180,E1 -5549.334,E2 -5549.334} C_VEL
LIN {X 0,Y 509.849,Z 142.48,A -85,B 0,C 180,E1 -5552.052,E2 -5552.052} C_VEL
LIN {X 0,Y 509.823,Z 142.475,A -85,B 0,C 180,E1 -5554.701,E2 -5554.701} C_VEL
LIN {X 0,Y 509.826,Z 142.477,A -85,B 0,C 180,E1 -5557.458,E2 -5557.458} C_VEL
LIN {X 0,Y 509.916,Z 142.472,A -85,B 0,C 180,E1 -5559.845,E2 -5559.845} C_VEL
LIN {X 0,Y 509.871,Z 142.47,A -85,B 0,C 180,E1 -5563.174,E2 -5563.174} C_VEL
LIN {X 0,Y 509.863,Z 142.478,A -85,B 0,C 180,E1 -5565.634,E2 -5565.634} C_VEL
LIN {X 0,Y 509.913,Z 142.464,A -85,B 0,C 180,E1 -5568.875,E2 -5568.875} C_VEL
LIN {X 0,Y 509.95,Z 142.46,A -85,B 0,C 180,E1 -5572.078,E2 -5572.078} C_VEL
LIN {X 0,Y 509.98,Z 142.455,A -85,B 0,C 180,E1 -5574.464,E2 -5574.464} C_VEL
LIN {X 0,Y 510.056,Z 142.449,A -85,B 0,C 180,E1 -5577.631,E2 -5577.631} C_VEL
LIN {X 0,Y 510.062,Z 142.448,A -85,B 0,C 180,E1 -5580.79,E2 -5580.79} C_VEL
LIN {X 0,Y 509.954,Z 142.467,A -85,B 0,C 180,E1 -5583.16,E2 -5583.16} C_VEL
LIN {X 0,Y 509.942,Z 142.46,A -85,B 0,C 180,E1 -5586.33,E2 -5586.33} C_VEL
LIN {X 0,Y 509.912,Z 142.468,A -85,B 0,C 180,E1 -5588.72,E2 -5588.72} C_VEL
LIN {X 0,Y 509.904,Z 142.464,A -85,B 0,C 180,E1 -5591.932,E2 -5591.932} C_VEL
LIN {X 0,Y 509.894,Z 142.468,A -85,B 0,C 180,E1 -5595.242,E2 -5595.242} C_VEL
LIN {X 0,Y 509.889,Z 142.467,A -85,B 0,C 180,E1 -5598.001,E2 -5598.001} C_VEL
LIN {X 0,Y 509.851,Z 142.474,A -85,B 0,C 180,E1 -5601.002,E2 -5601.002} C_VEL
LIN {X 0,Y 509.865,Z 142.477,A -85,B 0,C 180,E1 -5604.426,E2 -5604.426} C_VEL
LIN {X 0,Y 509.884,Z 142.468,A -85,B 0,C 180,E1 -5607.056,E2 -5607.056} C_VEL
LIN {X 0,Y 509.858,Z 142.472,A -85,B 0,C 180,E1 -5609.751,E2 -5609.751} C_VEL
LIN {X 0,Y 509.873,Z 142.47,A -85,B 0,C 180,E1 -5612.774,E2 -5612.774} C_VEL
LIN {X 0,Y 509.826,Z 142.475,A -85,B 0,C 180,E1 -5615.579,E2 -5615.579} C_VEL
LIN {X 0,Y 509.852,Z 142.476,A -85,B 0,C 180,E1 -5618.338,E2 -5618.338} C_VEL
LIN {X 0,Y 509.859,Z 142.472,A -85,B 0,C 180,E1 -5621.425,E2 -5621.425} C_VEL
LIN {X 0,Y 509.858,Z 142.47,A -85,B 0,C 180,E1 -5624.668,E2 -5624.668} C_VEL
LIN {X 0,Y 509.859,Z 142.474,A -85,B 0,C 180,E1 -5628.103,E2 -5628.103} C_VEL
LIN {X 0,Y 509.847,Z 142.471,A -85,B 0,C 180,E1 -5630.648,E2 -5630.648} C_VEL
LIN {X 0,Y 509.822,Z 142.482,A -85,B 0,C 180,E1 -5633.722,E2 -5633.722} C_VEL
LIN {X 0,Y 509.153,Z 142.56,A -85,B 0,C 180,E1 -5634.381,E2 -5634.381} C_VEL
LIN {X 0,Y 506.341,Z 142.915,A -85,B 0,C 180,E1 -5635.453,E2 -5635.453} C_VEL
LIN {X 0,Y 503.955,Z 143.21,A -85,B 0,C 180,E1 -5636.317,E2 -5636.317} C_VEL
LIN {X 0,Y 502.907,Z 143.338,A -85,B 0,C 180,E1 -5636.983,E2 -5636.983} C_VEL
LIN {X 0,Y 502.809,Z 143.349,A -85,B 0,C 180,E1 -5637.209,E2 -5637.209} C_VEL
LIN {X 0,Y 502.816,Z 143.348,A -85,B 0,C 180,E1 -5640.065,E2 -5640.065} C_VEL
LIN {X 0,Y 502.833,Z 143.345,A -85,B 0,C 180,E1 -5642.533,E2 -5642.533} C_VEL
LIN {X 0,Y 502.829,Z 143.353,A -85,B 0,C 180,E1 -5645.299,E2 -5645.299} C_VEL
LIN {X 0,Y 502.856,Z 143.425,A -85,B 0,C 180,E1 -5648.737,E2 -5648.737} C_VEL
LIN {X 0,Y 503.784,Z 149.735,A -85,B 0,C 180,E1 -5650.014,E2 -5650.014} C_VEL
LIN {X 0,Y 503.483,Z 162.914,A -85,B 0,C 180,E1 -5652.536,E2 -5652.536} C_VEL
LIN {X 0,Y 503.296,Z 172.227,A -85,B 0,C 180,E1 -5654.253,E2 -5654.253} C_VEL
LIN {X 0,Y 505.47,Z 184.399,A -85,B 0,C 180,E1 -5654.5,E2 -5654.5} C_VEL
LIN {X 0,Y 504.917,Z 279.562,A -85,B 0,C 180,E1 -5655.876,E2 -5655.876} C_VEL
LIN {X 0,Y 504.68,Z 292.719,A -85,B 0,C 180,E1 -5656.229,E2 -5656.229} C_VEL
LIN {X 0,Y 504.411,Z 304.807,A -85,B 0,C 180,E1 -5656.709,E2 -5656.709} C_VEL
LIN {X 0,Y 504.156,Z 316.397,A -85,B 0,C 180,E1 -5657.329,E2 -5657.329} C_VEL
LIN {X 0,Y 503.794,Z 327.887,A -85,B 0,C 180,E1 -5658.126,E2 -5658.126} C_VEL
LIN {X 0,Y 503.428,Z 338.367,A -85,B 0,C 180,E1 -5659.035,E2 -5659.035} C_VEL
LIN {X 0,Y 503.122,Z 346.929,A -85,B 0,C 180,E1 -5659.944,E2 -5659.944} C_VEL
LIN {X 0,Y 502.841,Z 354.815,A -85,B 0,C 180,E1 -5660.953,E2 -5660.953} C_VEL
LIN {X 0,Y 502.547,Z 362.528,A -85,B 0,C 180,E1 -5662.163,E2 -5662.163} C_VEL
LIN {X 0,Y 502.344,Z 369.601,A -85,B 0,C 180,E1 -5663.574,E2 -5663.574} C_VEL
LIN {X 0,Y 502.19,Z 374.316,A -85,B 0,C 180,E1 -5664.781,E2 -5664.781} C_VEL
LIN {X 0,Y 502.222,Z 377.924,A -85,B 0,C 180,E1 -5665.988,E2 -5665.988} C_VEL
LIN {X 0,Y 502.16,Z 379.791,A -85,B 0,C 180,E1 -5666.791,E2 -5666.791} C_VEL
LIN {X 0,Y 502.128,Z 381.199,A -85,B 0,C 180,E1 -5667.593,E2 -5667.593} C_VEL
LIN {X 0,Y 501.993,Z 382.82,A -85,B 0,C 180,E1 -5669.198,E2 -5669.198} C_VEL
LIN {X 0,Y 501.984,Z 383.057,A -85,B 0,C 180,E1 -5670,E2 -5670} C_VEL
LIN {X 0,Y 501.993,Z 382.873,A -85,B 0,C 180,E1 -5670.802,E2 -5670.802} C_VEL
LIN {X 0,Y 502.128,Z 381.322,A -85,B 0,C 180,E1 -5672.406,E2 -5672.406} C_VEL
LIN {X 0,Y 502.16,Z 379.966,A -85,B 0,C 180,E1 -5673.209,E2 -5673.209} C_VEL
LIN {X 0,Y 502.197,Z 377.102,A -85,B 0,C 180,E1 -5674.414,E2 -5674.414} C_VEL
LIN {X 0,Y 502.302,Z 373.216,A -85,B 0,C 180,E1 -5675.621,E2 -5675.621} C_VEL
LIN {X 0,Y 502.356,Z 368.205,A -85,B 0,C 180,E1 -5676.829,E2 -5676.829} C_VEL
LIN {X 0,Y 502.573,Z 361.894,A -85,B 0,C 180,E1 -5678.039,E2 -5678.039} C_VEL
LIN {X 0,Y 502.809,Z 353.995,A -85,B 0,C 180,E1 -5679.25,E2 -5679.25} C_VEL
LIN {X 0,Y 503.136,Z 345.941,A -85,B 0,C 180,E1 -5680.259,E2 -5680.259} C_VEL
LIN {X 0,Y 503.496,Z 336.114,A -85,B 0,C 180,E1 -5681.269,E2 -5681.269} C_VEL
LIN {X 0,Y 503.832,Z 326.448,A -85,B 0,C 180,E1 -5682.078,E2 -5682.078} C_VEL
LIN {X 0,Y 504.171,Z 315.471,A -85,B 0,C 180,E1 -5682.816,E2 -5682.816} C_VEL
LIN {X 0,Y 504.46,Z 303.418,A -85,B 0,C 180,E1 -5683.443,E2 -5683.443} C_VEL
LIN {X 0,Y 504.777,Z 290.068,A -85,B 0,C 180,E1 -5683.948,E2 -5683.948} C_VEL
LIN {X 0,Y 504.942,Z 277.586,A -85,B 0,C 180,E1 -5684.252,E2 -5684.252} C_VEL
LIN {X 0,Y 505.362,Z 183.626,A -85,B 0,C 180,E1 -5685.605,E2 -5685.605} C_VEL
LIN {X 0,Y 503.284,Z 172.022,A -85,B 0,C 180,E1 -5685.856,E2 -5685.856} C_VEL
LIN {X 0,Y 503.705,Z 154.586,A -85,B 0,C 180,E1 -5689.14,E2 -5689.14} C_VEL
LIN {X 0,Y 503.651,Z 148.024,A -85,B 0,C 180,E1 -5690.417,E2 -5690.417} C_VEL
LIN {X 0,Y 502.849,Z 143.351,A -85,B 0,C 180,E1 -5691.416,E2 -5691.416} C_VEL
LIN {X 0,Y 502.829,Z 143.353,A -85,B 0,C 180,E1 -5694.791,E2 -5694.791} C_VEL
LIN {X 0,Y 502.833,Z 143.346,A -85,B 0,C 180,E1 -5697.467,E2 -5697.467} C_VEL
LIN {X 0,Y 502.81,Z 143.351,A -85,B 0,C 180,E1 -5700.211,E2 -5700.211} C_VEL
LIN {X 0,Y 502.83,Z 143.348,A -85,B 0,C 180,E1 -5703.031,E2 -5703.031} C_VEL
LIN {X 0,Y 502.774,Z 143.355,A -85,B 0,C 180,E1 -5705.951,E2 -5705.951} C_VEL
LIN {X 0,Y 502.802,Z 143.35,A -85,B 0,C 180,E1 -5708.976,E2 -5708.976} C_VEL
LIN {X 0,Y 502.797,Z 143.356,A -85,B 0,C 180,E1 -5712.139,E2 -5712.139} C_VEL
LIN {X 0,Y 502.802,Z 143.35,A -85,B 0,C 180,E1 -5715.468,E2 -5715.468} C_VEL
LIN {X 0,Y 502.821,Z 143.347,A -85,B 0,C 180,E1 -5718.934,E2 -5718.934} C_VEL
LIN {X 0,Y 502.794,Z 143.358,A -85,B 0,C 180,E1 -5722.046,E2 -5722.046} C_VEL
LIN {X 0,Y 502.799,Z 143.35,A -85,B 0,C 180,E1 -5725.034,E2 -5725.034} C_VEL
LIN {X 0,Y 502.783,Z 143.358,A -85,B 0,C 180,E1 -5727.915,E2 -5727.915} C_VEL
LIN {X 0,Y 502.824,Z 143.346,A -85,B 0,C 180,E1 -5730.712,E2 -5730.712} C_VEL
LIN {X 0,Y 502.862,Z 143.347,A -85,B 0,C 180,E1 -5733.439,E2 -5733.439} C_VEL
LIN {X 0,Y 502.785,Z 143.353,A -85,B 0,C 180,E1 -5736.086,E2 -5736.086} C_VEL
LIN {X 0,Y 502.783,Z 143.352,A -85,B 0,C 180,E1 -5738.689,E2 -5738.689} C_VEL
LIN {X 0,Y 502.83,Z 143.352,A -85,B 0,C 180,E1 -5741.248,E2 -5741.248} C_VEL
LIN {X 0,Y 502.822,Z 143.349,A -85,B 0,C 180,E1 -5743.767,E2 -5743.767} C_VEL
LIN {X 0,Y 502.83,Z 143.345,A -85,B 0,C 180,E1 -5746.255,E2 -5746.255} C_VEL
LIN {X 0,Y 502.877,Z 143.342,A -85,B 0,C 180,E1 -5748.717,E2 -5748.717} C_VEL
LIN {X 0,Y 502.901,Z 143.337,A -85,B 0,C 180,E1 -5751.967,E2 -5751.967} C_VEL
LIN {X 0,Y 502.933,Z 143.334,A -85,B 0,C 180,E1 -5754.386,E2 -5754.386} C_VEL
LIN {X 0,Y 503.025,Z 143.322,A -85,B 0,C 180,E1 -5757.598,E2 -5757.598} C_VEL
LIN {X 0,Y 503.034,Z 143.329,A -85,B 0,C 180,E1 -5760.8,E2 -5760.8} C_VEL
LIN {X 0,Y 502.895,Z 143.34,A -85,B 0,C 180,E1 -5763.204,E2 -5763.204} C_VEL
LIN {X 0,Y 502.906,Z 143.342,A -85,B 0,C 180,E1 -5766.419,E2 -5766.419} C_VEL
LIN {X 0,Y 502.869,Z 143.345,A -85,B 0,C 180,E1 -5768.843,E2 -5768.843} C_VEL
LIN {X 0,Y 502.845,Z 143.347,A -85,B 0,C 180,E1 -5772.102,E2 -5772.102} C_VEL
LIN {X 0,Y 502.848,Z 143.343,A -85,B 0,C 180,E1 -5775.4,E2 -5775.4} C_VEL
LIN {X 0,Y 502.825,Z 143.348,A -85,B 0,C 180,E1 -5778.752,E2 -5778.752} C_VEL
LIN {X 0,Y 502.782,Z 143.352,A -85,B 0,C 180,E1 -5781.311,E2 -5781.311} C_VEL
LIN {X 0,Y 502.774,Z 143.359,A -85,B 0,C 180,E1 -5783.915,E2 -5783.915} C_VEL
LIN {X 0,Y 502.863,Z 143.343,A -85,B 0,C 180,E1 -5786.566,E2 -5786.566} C_VEL
LIN {X 0,Y 502.821,Z 143.348,A -85,B 0,C 180,E1 -5789.288,E2 -5789.288} C_VEL
LIN {X 0,Y 502.782,Z 143.356,A -85,B 0,C 180,E1 -5792.085,E2 -5792.085} C_VEL
LIN {X 0,Y 502.797,Z 143.35,A -85,B 0,C 180,E1 -5794.966,E2 -5794.966} C_VEL
LIN {X 0,Y 502.793,Z 143.35,A -85,B 0,C 180,E1 -5798.486,E2 -5798.486} C_VEL
LIN {X 0,Y 502.798,Z 143.352,A -85,B 0,C 180,E1 -5801.068,E2 -5801.068} C_VEL
LIN {X 0,Y 502.778,Z 143.352,A -85,B 0,C 180,E1 -5804.34,E2 -5804.34} C_VEL
LIN {X 0,Y 502.754,Z 143.356,A -85,B 0,C 180,E1 -5806.767,E2 -5806.767} C_VEL
LIN {X 0,Y 502.775,Z 143.357,A -85,B 0,C 180,E1 -5809.011,E2 -5809.011} C_VEL
LIN {X 0,Y 502.792,Z 143.351,A -85,B 0,C 180,E1 -5812.046,E2 -5812.046} C_VEL
LIN {X 0,Y 502.795,Z 143.357,A -85,B 0,C 180,E1 -5815.034,E2 -5815.034} C_VEL
LIN {X 0,Y 502.78,Z 143.352,A -85,B 0,C 180,E1 -5817.915,E2 -5817.915} C_VEL
LIN {X 0,Y 502.804,Z 143.356,A -85,B 0,C 180,E1 -5820.711,E2 -5820.711} C_VEL
LIN {X 0,Y 502.784,Z 143.356,A -85,B 0,C 180,E1 -5823.458,E2 -5823.458} C_VEL
LIN {X 0,Y 502.799,Z 143.391,A -85,B 0,C 180,E1 -5825.617,E2 -5825.617} C_VEL
LIN {X 0,Y 504.375,Z 152.386,A -85,B 0,C 180,E1 -5827.253,E2 -5827.253} C_VEL
LIN {X 0,Y 503.977,Z 166.16,A -85,B 0,C 180,E1 -5829.597,E2 -5829.597} C_VEL
LIN {X 0,Y 503.52,Z 182.413,A -85,B 0,C 180,E1 -5832.327,E2 -5832.327} C_VEL
LIN {X 0,Y 503.241,Z 193.636,A -85,B 0,C 180,E1 -5834.195,E2 -5834.195} C_VEL
LIN {X 0,Y 505.392,Z 207.533,A -85,B 0,C 180,E1 -5834.465,E2 -5834.465} C_VEL
LIN {X 0,Y 504.86,Z 301.656,A -85,B 0,C 180,E1 -5835.823,E2 -5835.823} C_VEL
LIN {X 0,Y 504.608,Z 314.936,A -85,B 0,C 180,E1 -5836.176,E2 -5836.176} C_VEL
LIN {X 0,Y 504.293,Z 327.102,A -85,B 0,C 180,E1 -5836.655,E2 -5836.655} C_VEL
LIN {X 0,Y 503.921,Z 339.182,A -85,B 0,C 180,E1 -5837.299,E2 -5837.299} C_VEL
LIN {X 0,Y 503.612,Z 349.679,A -85,B 0,C 180,E1 -5838.019,E2 -5838.019} C_VEL
LIN {X 0,Y 503.276,Z 360.343,A -85,B 0,C 180,E1 -5838.93,E2 -5838.93} C_VEL
LIN {X 0,Y 502.893,Z 369.949,A -85,B 0,C 180,E1 -5839.94,E2 -5839.94} C_VEL
LIN {X 0,Y 502.636,Z 377.825,A -85,B 0,C 180,E1 -5840.95,E2 -5840.95} C_VEL
LIN {X 0,Y 502.393,Z 385.516,A -85,B 0,C 180,E1 -5842.161,E2 -5842.161} C_VEL
LIN {X 0,Y 502.235,Z 392.606,A -85,B 0,C 180,E1 -5843.572,E2 -5843.572} C_VEL
LIN {X 0,Y 502.177,Z 397.323,A -85,B 0,C 180,E1 -5844.781,E2 -5844.781} C_VEL
LIN {X 0,Y 502.137,Z 400.926,A -85,B 0,C 180,E1 -5845.987,E2 -5845.987} C_VEL
LIN {X 0,Y 502.12,Z 402.785,A -85,B 0,C 180,E1 -5846.791,E2 -5846.791} C_VEL
LIN {X 0,Y 502.092,Z 404.178,A -85,B 0,C 180,E1 -5847.593,E2 -5847.593} C_VEL
LIN {X 0,Y 501.991,Z 405.777,A -85,B 0,C 180,E1 -5849.198,E2 -5849.198} C_VEL
LIN {X 0,Y 501.983,Z 405.993,A -85,B 0,C 180,E1 -5850,E2 -5850} C_VEL
LIN {X 0,Y 502.036,Z 405.173,A -85,B 0,C 180,E1 -5851.604,E2 -5851.604} C_VEL
LIN {X 0,Y 502.092,Z 404.181,A -85,B 0,C 180,E1 -5852.407,E2 -5852.407} C_VEL
LIN {X 0,Y 502.12,Z 402.788,A -85,B 0,C 180,E1 -5853.209,E2 -5853.209} C_VEL
LIN {X 0,Y 502.1,Z 399.857,A -85,B 0,C 180,E1 -5854.415,E2 -5854.415} C_VEL
LIN {X 0,Y 502.212,Z 395.891,A -85,B 0,C 180,E1 -5855.622,E2 -5855.622} C_VEL
LIN {X 0,Y 502.321,Z 389.89,A -85,B 0,C 180,E1 -5857.012,E2 -5857.012} C_VEL
LIN {X 0,Y 502.471,Z 383.12,A -85,B 0,C 180,E1 -5858.243,E2 -5858.243} C_VEL
LIN {X 0,Y 502.725,Z 374.845,A -85,B 0,C 180,E1 -5859.454,E2 -5859.454} C_VEL
LIN {X 0,Y 502.988,Z 366.363,A -85,B 0,C 180,E1 -5860.465,E2 -5860.465} C_VEL
LIN {X 0,Y 503.412,Z 355.884,A -85,B 0,C 180,E1 -5861.475,E2 -5861.475} C_VEL
LIN {X 0,Y 503.735,Z 344.299,A -85,B 0,C 180,E1 -5862.371,E2 -5862.371} C_VEL
LIN {X 0,Y 504.136,Z 332.224,A -85,B 0,C 180,E1 -5863.093,E2 -5863.093} C_VEL
LIN {X 0,Y 504.483,Z 319.883,A -85,B 0,C 180,E1 -5863.648,E2 -5863.648} C_VEL
LIN {X 0,Y 504.79,Z 307.22,A -85,B 0,C 180,E1 -5864.05,E2 -5864.05} C_VEL
LIN {X 0,Y 504.945,Z 294.003,A -85,B 0,C 180,E1 -5864.303,E2 -5864.303} C_VEL
LIN {X 0,Y 505.21,Z 206.081,A -85,B 0,C 180,E1 -5865.562,E2 -5865.562} C_VEL
LIN {X 0,Y 503.22,Z 193.556,A -85,B 0,C 180,E1 -5865.818,E2 -5865.818} C_VEL
LIN {X 0,Y 503.746,Z 174.911,A -85,B 0,C 180,E1 -5868.927,E2 -5868.927} C_VEL
LIN {X 0,Y 504.254,Z 158.643,A -85,B 0,C 180,E1 -5871.675,E2 -5871.675} C_VEL
LIN {X 0,Y 504.347,Z 151.122,A -85,B 0,C 180,E1 -5872.965,E2 -5872.965} C_VEL
LIN {X 0,Y 502.806,Z 143.356,A -85,B 0,C 180,E1 -5874.414,E2 -5874.414} C_VEL
LIN {X 0,Y 502.78,Z 143.355,A -85,B 0,C 180,E1 -5877.47,E2 -5877.47} C_VEL
LIN {X 0,Y 502.801,Z 143.348,A -85,B 0,C 180,E1 -5880.212,E2 -5880.212} C_VEL
LIN {X 0,Y 502.803,Z 143.356,A -85,B 0,C 180,E1 -5883.033,E2 -5883.033} C_VEL
LIN {X 0,Y 502.774,Z 143.353,A -85,B 0,C 180,E1 -5885.951,E2 -5885.951} C_VEL
LIN {X 0,Y 502.793,Z 143.355,A -85,B 0,C 180,E1 -5888.977,E2 -5888.977} C_VEL
LIN {X 0,Y 502.804,Z 143.351,A -85,B 0,C 180,E1 -5892.199,E2 -5892.199} C_VEL
LIN {X 0,Y 502.785,Z 143.351,A -85,B 0,C 180,E1 -5895.47,E2 -5895.47} C_VEL
LIN {X 0,Y 502.795,Z 143.351,A -85,B 0,C 180,E1 -5897.86,E2 -5897.86} C_VEL
LIN {X 0,Y 502.801,Z 143.35,A -85,B 0,C 180,E1 -5901.024,E2 -5901.024} C_VEL
LIN {X 0,Y 502.771,Z 143.36,A -85,B 0,C 180,E1 -5904.17,E2 -5904.17} C_VEL
LIN {X 0,Y 502.832,Z 143.346,A -85,B 0,C 180,E1 -5906.993,E2 -5906.993} C_VEL
LIN {X 0,Y 502.814,Z 143.355,A -85,B 0,C 180,E1 -5910.065,E2 -5910.065} C_VEL
LIN {X 0,Y 502.844,Z 143.345,A -85,B 0,C 180,E1 -5913.443,E2 -5913.443} C_VEL
LIN {X 0,Y 502.774,Z 143.359,A -85,B 0,C 180,E1 -5916.085,E2 -5916.085} C_VEL
LIN {X 0,Y 502.783,Z 143.352,A -85,B 0,C 180,E1 -5918.689,E2 -5918.689} C_VEL
LIN {X 0,Y 502.825,Z 143.348,A -85,B 0,C 180,E1 -5921.248,E2 -5921.248} C_VEL
LIN {X 0,Y 502.848,Z 143.343,A -85,B 0,C 180,E1 -5924.6,E2 -5924.6} C_VEL
LIN {X 0,Y 502.876,Z 143.342,A -85,B 0,C 180,E1 -5928.039,E2 -5928.039} C_VEL
LIN {X 0,Y 502.869,Z 143.345,A -85,B 0,C 180,E1 -5931.157,E2 -5931.157} C_VEL
LIN {X 0,Y 502.906,Z 143.342,A -85,B 0,C 180,E1 -5933.581,E2 -5933.581} C_VEL
LIN {X 0,Y 502.895,Z 143.339,A -85,B 0,C 180,E1 -5936.796,E2 -5936.796} C_VEL
LIN {X 0,Y 503.034,Z 143.328,A -85,B 0,C 180,E1 -5939.2,E2 -5939.2} C_VEL
LIN {X 0,Y 503.025,Z 143.322,A -85,B 0,C 180,E1 -5942.402,E2 -5942.402} C_VEL
LIN {X 0,Y 502.93,Z 143.335,A -85,B 0,C 180,E1 -5945.614,E2 -5945.614} C_VEL
LIN {X 0,Y 502.87,Z 143.347,A -85,B 0,C 180,E1 -5948.843,E2 -5948.843} C_VEL
LIN {X 0,Y 502.846,Z 143.344,A -85,B 0,C 180,E1 -5952.102,E2 -5952.102} C_VEL
LIN {X 0,Y 502.849,Z 143.344,A -85,B 0,C 180,E1 -5955.4,E2 -5955.4} C_VEL
LIN {X 0,Y 502.846,Z 143.345,A -85,B 0,C 180,E1 -5958.122,E2 -5958.122} C_VEL
LIN {X 0,Y 502.829,Z 143.353,A -85,B 0,C 180,E1 -5960.536,E2 -5960.536} C_VEL
LIN {X 0,Y 502.791,Z 143.353,A -85,B 0,C 180,E1 -5963.041,E2 -5963.041} C_VEL
LIN {X 0,Y 502.84,Z 143.345,A -85,B 0,C 180,E1 -5965.676,E2 -5965.676} C_VEL
LIN {X 0,Y 502.84,Z 143.353,A -85,B 0,C 180,E1 -5968.373,E2 -5968.373} C_VEL
LIN {X 0,Y 502.793,Z 143.35,A -85,B 0,C 180,E1 -5971.499,E2 -5971.499} C_VEL
LIN {X 0,Y 502.804,Z 143.354,A -85,B 0,C 180,E1 -5973.994,E2 -5973.994} C_VEL
LIN {X 0,Y 502.778,Z 143.352,A -85,B 0,C 180,E1 -5977.178,E2 -5977.178} C_VEL
LIN {X 0,Y 502.789,Z 143.359,A -85,B 0,C 180,E1 -5980.015,E2 -5980.015} C_VEL
LIN {X 0,Y 502.804,Z 143.354,A -85,B 0,C 180,E1 -5982.199,E2 -5982.199} C_VEL
LIN {X 0,Y 502.802,Z 143.352,A -85,B 0,C 180,E1 -5985.468,E2 -5985.468} C_VEL
LIN {X 0,Y 502.821,Z 143.347,A -85,B 0,C 180,E1 -5988.934,E2 -5988.934} C_VEL
LIN {X 0,Y 502.795,Z 143.353,A -85,B 0,C 180,E1 -5992.046,E2 -5992.046} C_VEL
LIN {X 0,Y 502.797,Z 143.351,A -85,B 0,C 180,E1 -5995.034,E2 -5995.034} C_VEL
LIN {X 0,Y 502.809,Z 143.349,A -85,B 0,C 180,E1 -5997.209,E2 -5997.209} C_VEL
LIN {X 0,Y 502.107,Z 143.439,A -85,B 0,C 180,E1 -5997.877,E2 -5997.877} C_VEL
LIN {X 0,Y 499.243,Z 143.794,A -85,B 0,C 180,E1 -5998.963,E2 -5998.963} C_VEL
LIN {X 0,Y 496.85,Z 144.094,A -85,B 0,C 180,E1 -5999.838,E2 -5999.838} C_VEL
LIN {X 0,Y 495.833,Z 144.218,A -85,B 0,C 180,E1 -6000.514,E2 -6000.514} C_VEL
LIN {X 0,Y 495.754,Z 144.228,A -85,B 0,C 180,E1 -6000.742,E2 -6000.742} C_VEL
LIN {X 0,Y 495.793,Z 144.225,A -85,B 0,C 180,E1 -6003.932,E2 -6003.932} C_VEL
LIN {X 0,Y 495.763,Z 144.233,A -85,B 0,C 180,E1 -6007.14,E2 -6007.14} C_VEL
LIN {X 0,Y 495.799,Z 144.336,A -85,B 0,C 180,E1 -6008.592,E2 -6008.592} C_VEL
LIN {X 0,Y 496.826,Z 150.895,A -85,B 0,C 180,E1 -6009.938,E2 -6009.938} C_VEL
LIN {X 0,Y 496.507,Z 164.137,A -85,B 0,C 180,E1 -6012.495,E2 -6012.495} C_VEL
LIN {X 0,Y 496.339,Z 172.225,A -85,B 0,C 180,E1 -6014.02,E2 -6014.02} C_VEL
LIN {X 0,Y 498.604,Z 184.786,A -85,B 0,C 180,E1 -6014.284,E2 -6014.284} C_VEL
LIN {X 0,Y 498.062,Z 279.745,A -85,B 0,C 180,E1 -6015.678,E2 -6015.678} C_VEL
LIN {X 0,Y 497.811,Z 292.895,A -85,B 0,C 180,E1 -6016.035,E2 -6016.035} C_VEL
LIN {X 0,Y 497.515,Z 304.98,A -85,B 0,C 180,E1 -6016.521,E2 -6016.521} C_VEL
LIN {X 0,Y 497.216,Z 315.605,A -85,B 0,C 180,E1 -6017.091,E2 -6017.091} C_VEL
LIN {X 0,Y 496.871,Z 326.769,A -85,B 0,C 180,E1 -6017.854,E2 -6017.854} C_VEL
LIN {X 0,Y 496.478,Z 337.469,A -85,B 0,C 180,E1 -6018.776,E2 -6018.776} C_VEL
LIN {X 0,Y 496.124,Z 347.096,A -85,B 0,C 180,E1 -6019.801,E2 -6019.801} C_VEL
LIN {X 0,Y 495.801,Z 354.982,A -85,B 0,C 180,E1 -6020.824,E2 -6020.824} C_VEL
LIN {X 0,Y 495.515,Z 362.693,A -85,B 0,C 180,E1 -6022.051,E2 -6022.051} C_VEL
LIN {X 0,Y 495.273,Z 369.766,A -85,B 0,C 180,E1 -6023.482,E2 -6023.482} C_VEL
LIN {X 0,Y 495.132,Z 374.48,A -85,B 0,C 180,E1 -6024.706,E2 -6024.706} C_VEL
LIN {X 0,Y 495.14,Z 378.088,A -85,B 0,C 180,E1 -6025.93,E2 -6025.93} C_VEL
LIN {X 0,Y 495.082,Z 379.954,A -85,B 0,C 180,E1 -6026.745,E2 -6026.745} C_VEL
LIN {X 0,Y 495.033,Z 381.363,A -85,B 0,C 180,E1 -6027.559,E2 -6027.559} C_VEL
LIN {X 0,Y 494.913,Z 382.982,A -85,B 0,C 180,E1 -6029.186,E2 -6029.186} C_VEL
LIN {X 0,Y 494.902,Z 383.219,A -85,B 0,C 180,E1 -6030,E2 -6030} C_VEL
LIN {X 0,Y 494.913,Z 383.034,A -85,B 0,C 180,E1 -6030.814,E2 -6030.814} C_VEL
LIN {X 0,Y 495.033,Z 381.483,A -85,B 0,C 180,E1 -6032.441,E2 -6032.441} C_VEL
LIN {X 0,Y 495.082,Z 380.127,A -85,B 0,C 180,E1 -6033.255,E2 -6033.255} C_VEL
LIN {X 0,Y 495.092,Z 377.263,A -85,B 0,C 180,E1 -6034.478,E2 -6034.478} C_VEL
LIN {X 0,Y 495.251,Z 373.375,A -85,B 0,C 180,E1 -6035.701,E2 -6035.701} C_VEL
LIN {X 0,Y 495.308,Z 368.365,A -85,B 0,C 180,E1 -6036.927,E2 -6036.927} C_VEL
LIN {X 0,Y 495.529,Z 362.054,A -85,B 0,C 180,E1 -6038.154,E2 -6038.154} C_VEL
LIN {X 0,Y 495.794,Z 354.153,A -85,B 0,C 180,E1 -6039.382,E2 -6039.382} C_VEL
LIN {X 0,Y 496.113,Z 346.1,A -85,B 0,C 180,E1 -6040.406,E2 -6040.406} C_VEL
LIN {X 0,Y 496.534,Z 336.271,A -85,B 0,C 180,E1 -6041.429,E2 -6041.429} C_VEL
LIN {X 0,Y 496.918,Z 325.245,A -85,B 0,C 180,E1 -6042.351,E2 -6042.351} C_VEL
LIN {X 0,Y 497.266,Z 314.397,A -85,B 0,C 180,E1 -6043.069,E2 -6043.069} C_VEL
LIN {X 0,Y 497.587,Z 302.441,A -85,B 0,C 180,E1 -6043.685,E2 -6043.685} C_VEL
LIN {X 0,Y 497.934,Z 289.352,A -85,B 0,C 180,E1 -6044.17,E2 -6044.17} C_VEL
LIN {X 0,Y 498.092,Z 276.215,A -85,B 0,C 180,E1 -6044.478,E2 -6044.478} C_VEL
LIN {X 0,Y 498.549,Z 184.372,A -85,B 0,C 180,E1 -6045.815,E2 -6045.815} C_VEL
LIN {X 0,Y 496.302,Z 172.207,A -85,B 0,C 180,E1 -6046.076,E2 -6046.076} C_VEL
LIN {X 0,Y 496.736,Z 155.764,A -85,B 0,C 180,E1 -6049.205,E2 -6049.205} C_VEL
LIN {X 0,Y 496.681,Z 149.174,A -85,B 0,C 180,E1 -6050.5,E2 -6050.5} C_VEL
LIN {X 0,Y 495.805,Z 144.227,A -85,B 0,C 180,E1 -6051.544,E2 -6051.544} C_VEL
LIN {X 0,Y 495.79,Z 144.228,A -85,B 0,C 180,E1 -6055.167,E2 -6055.167} C_VEL
LIN {X 0,Y 495.781,Z 144.224,A -85,B 0,C 180,E1 -6057.891,E2 -6057.891} C_VEL
LIN {X 0,Y 495.752,Z 144.235,A -85,B 0,C 180,E1 -6060.687,E2 -6060.687} C_VEL
LIN {X 0,Y 495.752,Z 144.227,A -85,B 0,C 180,E1 -6063.565,E2 -6063.565} C_VEL
LIN {X 0,Y 495.729,Z 144.237,A -85,B 0,C 180,E1 -6066.544,E2 -6066.544} C_VEL
LIN {X 0,Y 495.757,Z 144.227,A -85,B 0,C 180,E1 -6069.638,E2 -6069.638} C_VEL
LIN {X 0,Y 495.738,Z 144.234,A -85,B 0,C 180,E1 -6072.507,E2 -6072.507} C_VEL
LIN {X 0,Y 495.75,Z 144.227,A -85,B 0,C 180,E1 -6075.139,E2 -6075.139} C_VEL
LIN {X 0,Y 495.757,Z 144.233,A -85,B 0,C 180,E1 -6078.219,E2 -6078.219} C_VEL
LIN {X 0,Y 495.751,Z 144.229,A -85,B 0,C 180,E1 -6081.408,E2 -6081.408} C_VEL
LIN {X 0,Y 495.748,Z 144.229,A -85,B 0,C 180,E1 -6084.462,E2 -6084.462} C_VEL
LIN {X 0,Y 495.767,Z 144.228,A -85,B 0,C 180,E1 -6087.405,E2 -6087.405} C_VEL
LIN {X 0,Y 495.766,Z 144.227,A -85,B 0,C 180,E1 -6090.253,E2 -6090.253} C_VEL
LIN {X 0,Y 495.823,Z 144.222,A -85,B 0,C 180,E1 -6093.251,E2 -6093.251} C_VEL
LIN {X 0,Y 495.748,Z 144.234,A -85,B 0,C 180,E1 -6095.725,E2 -6095.725} C_VEL
LIN {X 0,Y 495.742,Z 144.229,A -85,B 0,C 180,E1 -6098.371,E2 -6098.371} C_VEL
LIN {X 0,Y 495.784,Z 144.226,A -85,B 0,C 180,E1 -6100.971,E2 -6100.971} C_VEL
LIN {X 0,Y 495.779,Z 144.229,A -85,B 0,C 180,E1 -6103.53,E2 -6103.53} C_VEL
LIN {X 0,Y 495.793,Z 144.222,A -85,B 0,C 180,E1 -6106.056,E2 -6106.056} C_VEL
LIN {X 0,Y 495.851,Z 144.216,A -85,B 0,C 180,E1 -6108.555,E2 -6108.555} C_VEL
LIN {X 0,Y 495.872,Z 144.213,A -85,B 0,C 180,E1 -6111.852,E2 -6111.852} C_VEL
LIN {X 0,Y 495.889,Z 144.211,A -85,B 0,C 180,E1 -6114.306,E2 -6114.306} C_VEL
LIN {X 0,Y 495.993,Z 144.198,A -85,B 0,C 180,E1 -6117.564,E2 -6117.564} C_VEL
LIN {X 0,Y 496.004,Z 144.204,A -85,B 0,C 180,E1 -6120.812,E2 -6120.812} C_VEL
LIN {X 0,Y 495.839,Z 144.218,A -85,B 0,C 180,E1 -6123.25,E2 -6123.25} C_VEL
LIN {X 0,Y 495.86,Z 144.221,A -85,B 0,C 180,E1 -6126.511,E2 -6126.511} C_VEL
LIN {X 0,Y 495.838,Z 144.219,A -85,B 0,C 180,E1 -6128.97,E2 -6128.97} C_VEL
LIN {X 0,Y 495.827,Z 144.221,A -85,B 0,C 180,E1 -6132.035,E2 -6132.035} C_VEL
LIN {X 0,Y 495.823,Z 144.219,A -85,B 0,C 180,E1 -6135.452,E2 -6135.452} C_VEL
LIN {X 0,Y 495.778,Z 144.233,A -85,B 0,C 180,E1 -6138.237,E2 -6138.237} C_VEL
LIN {X 0,Y 495.773,Z 144.226,A -85,B 0,C 180,E1 -6140.756,E2 -6140.756} C_VEL
LIN {X 0,Y 495.742,Z 144.229,A -85,B 0,C 180,E1 -6143.388,E2 -6143.388} C_VEL
LIN {X 0,Y 495.822,Z 144.219,A -85,B 0,C 180,E1 -6146.749,E2 -6146.749} C_VEL
LIN {X 0,Y 495.765,Z 144.232,A -85,B 0,C 180,E1 -6149.747,E2 -6149.747} C_VEL
LIN {X 0,Y 495.767,Z 144.226,A -85,B 0,C 180,E1 -6152.595,E2 -6152.595} C_VEL
LIN {X 0,Y 495.744,Z 144.234,A -85,B 0,C 180,E1 -6155.538,E2 -6155.538} C_VEL
LIN {X 0,Y 495.762,Z 144.226,A -85,B 0,C 180,E1 -6158.768,E2 -6158.768} C_VEL
LIN {X 0,Y 495.75,Z 144.233,A -85,B 0,C 180,E1 -6161.782,E2 -6161.782} C_VEL
LIN {X 0,Y 495.737,Z 144.233,A -85,B 0,C 180,E1 -6165.141,E2 -6165.141} C_VEL
LIN {X 0,Y 495.744,Z 144.228,A -85,B 0,C 180,E1 -6168.218,E2 -6168.218} C_VEL
LIN {X 0,Y 495.746,Z 144.234,A -85,B 0,C 180,E1 -6171.408,E2 -6171.408} C_VEL
LIN {X 0,Y 495.747,Z 144.229,A -85,B 0,C 180,E1 -6174.462,E2 -6174.462} C_VEL
LIN {X 0,Y 495.765,Z 144.229,A -85,B 0,C 180,E1 -6177.406,E2 -6177.406} C_VEL
LIN {X 0,Y 495.757,Z 144.23,A -85,B 0,C 180,E1 -6180.253,E2 -6180.253} C_VEL
LIN {X 0,Y 495.742,Z 144.233,A -85,B 0,C 180,E1 -6183.27,E2 -6183.27} C_VEL
LIN {X 0,Y 495.79,Z 144.32,A -85,B 0,C 180,E1 -6185.443,E2 -6185.443} C_VEL
LIN {X 0,Y 497.429,Z 153.566,A -85,B 0,C 180,E1 -6187.151,E2 -6187.151} C_VEL
LIN {X 0,Y 496.999,Z 168.505,A -85,B 0,C 180,E1 -6189.73,E2 -6189.73} C_VEL
LIN {X 0,Y 496.464,Z 186,A -85,B 0,C 180,E1 -6192.706,E2 -6192.706} C_VEL
LIN {X 0,Y 496.229,Z 193.461,A -85,B 0,C 180,E1 -6193.964,E2 -6193.964} C_VEL
LIN {X 0,Y 498.543,Z 209.038,A -85,B 0,C 180,E1 -6194.27,E2 -6194.27} C_VEL
LIN {X 0,Y 497.99,Z 301.501,A -85,B 0,C 180,E1 -6195.623,E2 -6195.623} C_VEL
LIN {X 0,Y 497.727,Z 314.778,A -85,B 0,C 180,E1 -6195.981,E2 -6195.981} C_VEL
LIN {X 0,Y 497.371,Z 326.943,A -85,B 0,C 180,E1 -6196.465,E2 -6196.465} C_VEL
LIN {X 0,Y 496.977,Z 339.312,A -85,B 0,C 180,E1 -6197.137,E2 -6197.137} C_VEL
LIN {X 0,Y 496.617,Z 350.813,A -85,B 0,C 180,E1 -6197.952,E2 -6197.952} C_VEL
LIN {X 0,Y 496.249,Z 361.253,A -85,B 0,C 180,E1 -6198.874,E2 -6198.874} C_VEL
LIN {X 0,Y 495.851,Z 369.787,A -85,B 0,C 180,E1 -6199.795,E2 -6199.795} C_VEL
LIN {X 0,Y 495.601,Z 377.663,A -85,B 0,C 180,E1 -6200.82,E2 -6200.82} C_VEL
LIN {X 0,Y 495.335,Z 385.353,A -85,B 0,C 180,E1 -6202.048,E2 -6202.048} C_VEL
LIN {X 0,Y 495.164,Z 392.443,A -85,B 0,C 180,E1 -6203.48,E2 -6203.48} C_VEL
LIN {X 0,Y 495.109,Z 397.161,A -85,B 0,C 180,E1 -6204.706,E2 -6204.706} C_VEL
LIN {X 0,Y 495.031,Z 400.764,A -85,B 0,C 180,E1 -6205.929,E2 -6205.929} C_VEL
LIN {X 0,Y 495.041,Z 402.623,A -85,B 0,C 180,E1 -6206.745,E2 -6206.745} C_VEL
LIN {X 0,Y 494.998,Z 404.016,A -85,B 0,C 180,E1 -6207.559,E2 -6207.559} C_VEL
LIN {X 0,Y 494.962,Z 405.01,A -85,B 0,C 180,E1 -6208.373,E2 -6208.373} C_VEL
LIN {X 0,Y 494.901,Z 405.832,A -85,B 0,C 180,E1 -6210,E2 -6210} C_VEL
LIN {X 0,Y 494.962,Z 405.011,A -85,B 0,C 180,E1 -6211.627,E2 -6211.627} C_VEL
LIN {X 0,Y 494.998,Z 404.019,A -85,B 0,C 180,E1 -6212.441,E2 -6212.441} C_VEL
LIN {X 0,Y 495.041,Z 402.626,A -85,B 0,C 180,E1 -6213.255,E2 -6213.255} C_VEL
LIN {X 0,Y 495.006,Z 399.694,A -85,B 0,C 180,E1 -6214.479,E2 -6214.479} C_VEL
LIN {X 0,Y 495.126,Z 395.728,A -85,B 0,C 180,E1 -6215.702,E2 -6215.702} C_VEL
LIN {X 0,Y 495.251,Z 389.626,A -85,B 0,C 180,E1 -6217.133,E2 -6217.133} C_VEL
LIN {X 0,Y 495.418,Z 382.957,A -85,B 0,C 180,E1 -6218.361,E2 -6218.361} C_VEL
LIN {X 0,Y 495.709,Z 374.682,A -85,B 0,C 180,E1 -6219.589,E2 -6219.589} C_VEL
LIN {X 0,Y 495.984,Z 366.199,A -85,B 0,C 180,E1 -6220.615,E2 -6220.615} C_VEL
LIN {X 0,Y 496.449,Z 355.72,A -85,B 0,C 180,E1 -6221.638,E2 -6221.638} C_VEL
LIN {X 0,Y 496.77,Z 344.343,A -85,B 0,C 180,E1 -6222.532,E2 -6222.532} C_VEL
LIN {X 0,Y 497.206,Z 332.058,A -85,B 0,C 180,E1 -6223.279,E2 -6223.279} C_VEL
LIN {X 0,Y 497.587,Z 319.717,A -85,B 0,C 180,E1 -6223.841,E2 -6223.841} C_VEL
LIN {X 0,Y 497.918,Z 307.052,A -85,B 0,C 180,E1 -6224.248,E2 -6224.248} C_VEL
LIN {X 0,Y 498.07,Z 293.829,A -85,B 0,C 180,E1 -6224.505,E2 -6224.505} C_VEL
LIN {X 0,Y 498.502,Z 207.572,A -85,B 0,C 180,E1 -6225.752,E2 -6225.752} C_VEL
LIN {X 0,Y 496.228,Z 193.456,A -85,B 0,C 180,E1 -6226.036,E2 -6226.036} C_VEL
LIN {X 0,Y 496.801,Z 174.749,A -85,B 0,C 180,E1 -6229.202,E2 -6229.202} C_VEL
LIN {X 0,Y 497.304,Z 159.735,A -85,B 0,C 180,E1 -6231.775,E2 -6231.775} C_VEL
LIN {X 0,Y 497.476,Z 153.538,A -85,B 0,C 180,E1 -6232.849,E2 -6232.849} C_VEL
LIN {X 0,Y 495.761,Z 144.234,A -85,B 0,C 180,E1 -6234.58,E2 -6234.58} C_VEL
LIN {X 0,Y 495.719,Z 144.231,A -85,B 0,C 180,E1 -6237.895,E2 -6237.895} C_VEL
LIN {X 0,Y 495.744,Z 144.231,A -85,B 0,C 180,E1 -6240.688,E2 -6240.688} C_VEL
LIN {X 0,Y 495.742,Z 144.23,A -85,B 0,C 180,E1 -6243.566,E2 -6243.566} C_VEL
LIN {X 0,Y 495.728,Z 144.235,A -85,B 0,C 180,E1 -6246.544,E2 -6246.544} C_VEL
LIN {X 0,Y 495.744,Z 144.228,A -85,B 0,C 180,E1 -6249.639,E2 -6249.639} C_VEL
LIN {X 0,Y 495.715,Z 144.237,A -85,B 0,C 180,E1 -6252.884,E2 -6252.884} C_VEL
LIN {X 0,Y 495.725,Z 144.232,A -85,B 0,C 180,E1 -6255.998,E2 -6255.998} C_VEL
LIN {X 0,Y 495.739,Z 144.234,A -85,B 0,C 180,E1 -6258.709,E2 -6258.709} C_VEL
LIN {X 0,Y 495.749,Z 144.228,A -85,B 0,C 180,E1 -6261.408,E2 -6261.408} C_VEL
LIN {X 0,Y 495.745,Z 144.234,A -85,B 0,C 180,E1 -6264.462,E2 -6264.462} C_VEL
LIN {X 0,Y 495.767,Z 144.226,A -85,B 0,C 180,E1 -6267.406,E2 -6267.406} C_VEL
LIN {X 0,Y 495.762,Z 144.233,A -85,B 0,C 180,E1 -6270.253,E2 -6270.253} C_VEL
LIN {X 0,Y 495.774,Z 144.225,A -85,B 0,C 180,E1 -6273.262,E2 -6273.262} C_VEL
LIN {X 0,Y 495.742,Z 144.229,A -85,B 0,C 180,E1 -6276.612,E2 -6276.612} C_VEL
LIN {X 0,Y 495.778,Z 144.226,A -85,B 0,C 180,E1 -6279.324,E2 -6279.324} C_VEL
LIN {X 0,Y 495.78,Z 144.232,A -85,B 0,C 180,E1 -6281.828,E2 -6281.828} C_VEL
LIN {X 0,Y 495.823,Z 144.219,A -85,B 0,C 180,E1 -6284.548,E2 -6284.548} C_VEL
LIN {X 0,Y 495.828,Z 144.221,A -85,B 0,C 180,E1 -6287.965,E2 -6287.965} C_VEL
LIN {X 0,Y 495.838,Z 144.219,A -85,B 0,C 180,E1 -6291.03,E2 -6291.03} C_VEL
LIN {X 0,Y 495.861,Z 144.221,A -85,B 0,C 180,E1 -6293.489,E2 -6293.489} C_VEL
LIN {X 0,Y 495.839,Z 144.218,A -85,B 0,C 180,E1 -6296.75,E2 -6296.75} C_VEL
LIN {X 0,Y 496.005,Z 144.203,A -85,B 0,C 180,E1 -6299.188,E2 -6299.188} C_VEL
LIN {X 0,Y 495.993,Z 144.198,A -85,B 0,C 180,E1 -6302.436,E2 -6302.436} C_VEL
LIN {X 0,Y 495.885,Z 144.212,A -85,B 0,C 180,E1 -6305.694,E2 -6305.694} C_VEL
LIN {X 0,Y 495.839,Z 144.225,A -85,B 0,C 180,E1 -6308.97,E2 -6308.97} C_VEL
LIN {X 0,Y 495.828,Z 144.218,A -85,B 0,C 180,E1 -6312.035,E2 -6312.035} C_VEL
LIN {X 0,Y 495.824,Z 144.219,A -85,B 0,C 180,E1 -6315.452,E2 -6315.452} C_VEL
LIN {X 0,Y 495.807,Z 144.223,A -85,B 0,C 180,E1 -6318.247,E2 -6318.247} C_VEL
LIN {X 0,Y 495.774,Z 144.231,A -85,B 0,C 180,E1 -6320.757,E2 -6320.757} C_VEL
LIN {X 0,Y 495.748,Z 144.228,A -85,B 0,C 180,E1 -6323.387,E2 -6323.387} C_VEL
LIN {X 0,Y 495.791,Z 144.226,A -85,B 0,C 180,E1 -6326.068,E2 -6326.068} C_VEL
LIN {X 0,Y 495.772,Z 144.227,A -85,B 0,C 180,E1 -6328.815,E2 -6328.815} C_VEL
LIN {X 0,Y 495.755,Z 144.229,A -85,B 0,C 180,E1 -6331.725,E2 -6331.725} C_VEL
LIN {X 0,Y 495.769,Z 144.227,A -85,B 0,C 180,E1 -6334.694,E2 -6334.694} C_VEL
LIN {X 0,Y 495.73,Z 144.232,A -85,B 0,C 180,E1 -6337.562,E2 -6337.562} C_VEL
LIN {X 0,Y 495.768,Z 144.226,A -85,B 0,C 180,E1 -6340.7,E2 -6340.7} C_VEL
LIN {X 0,Y 495.735,Z 144.237,A -85,B 0,C 180,E1 -6344.001,E2 -6344.001} C_VEL
LIN {X 0,Y 495.727,Z 144.231,A -85,B 0,C 180,E1 -6347.117,E2 -6347.117} C_VEL
LIN {X 0,Y 495.76,Z 144.232,A -85,B 0,C 180,E1 -6349.953,E2 -6349.953} C_VEL
LIN {X 0,Y 495.729,Z 144.23,A -85,B 0,C 180,E1 -6352.553,E2 -6352.553} C_VEL
LIN {X 0,Y 495.772,Z 144.232,A -85,B 0,C 180,E1 -6355.456,E2 -6355.456} C_VEL
LIN {X 0,Y 495.756,Z 144.227,A -85,B 0,C 180,E1 -6358.364,E2 -6358.364} C_VEL
LIN {X 0,Y 495.754,Z 144.228,A -85,B 0,C 180,E1 -6360.742,E2 -6360.742} C_VEL
LIN {X 0,Y 495.096,Z 144.317,A -85,B 0,C 180,E1 -6361.421,E2 -6361.421} C_VEL
LIN {X 0,Y 492.241,Z 144.669,A -85,B 0,C 180,E1 -6362.524,E2 -6362.524} C_VEL
LIN {X 0,Y 489.833,Z 144.973,A -85,B 0,C 180,E1 -6363.413,E2 -6363.413} C_VEL
LIN {X 0,Y 488.817,Z 145.094,A -85,B 0,C 180,E1 -6364.099,E2 -6364.099} C_VEL
LIN {X 0,Y 488.744,Z 145.102,A -85,B 0,C 180,E1 -6364.331,E2 -6364.331} C_VEL
LIN {X 0,Y 488.725,Z 145.109,A -85,B 0,C 180,E1 -6367.153,E2 -6367.153} C_VEL
LIN {X 0,Y 488.757,Z 145.215,A -85,B 0,C 180,E1 -6368.434,E2 -6368.434} C_VEL
LIN {X 0,Y 489.857,Z 152.073,A -85,B 0,C 180,E1 -6369.859,E2 -6369.859} C_VEL
LIN {X 0,Y 489.533,Z 165.377,A -85,B 0,C 180,E1 -6372.453,E2 -6372.453} C_VEL
LIN {X 0,Y 489.354,Z 172.414,A -85,B 0,C 180,E1 -6373.789,E2 -6373.789} C_VEL
LIN {X 0,Y 491.823,Z 186.586,A -85,B 0,C 180,E1 -6374.085,E2 -6374.085} C_VEL
LIN {X 0,Y 491.215,Z 279.926,A -85,B 0,C 180,E1 -6375.474,E2 -6375.474} C_VEL
LIN {X 0,Y 490.916,Z 293.831,A -85,B 0,C 180,E1 -6375.861,E2 -6375.861} C_VEL
LIN {X 0,Y 490.604,Z 306.263,A -85,B 0,C 180,E1 -6376.381,E2 -6376.381} C_VEL
LIN {X 0,Y 490.284,Z 317.757,A -85,B 0,C 180,E1 -6377.032,E2 -6377.032} C_VEL
LIN {X 0,Y 489.909,Z 328.224,A -85,B 0,C 180,E1 -6377.784,E2 -6377.784} C_VEL
LIN {X 0,Y 489.489,Z 338.701,A -85,B 0,C 180,E1 -6378.719,E2 -6378.719} C_VEL
LIN {X 0,Y 489.13,Z 347.262,A -85,B 0,C 180,E1 -6379.653,E2 -6379.653} C_VEL
LIN {X 0,Y 488.764,Z 355.148,A -85,B 0,C 180,E1 -6380.691,E2 -6380.691} C_VEL
LIN {X 0,Y 488.47,Z 362.858,A -85,B 0,C 180,E1 -6381.936,E2 -6381.936} C_VEL
LIN {X 0,Y 488.222,Z 369.93,A -85,B 0,C 180,E1 -6383.387,E2 -6383.387} C_VEL
LIN {X 0,Y 488.078,Z 374.643,A -85,B 0,C 180,E1 -6384.629,E2 -6384.629} C_VEL
LIN {X 0,Y 488.043,Z 378.252,A -85,B 0,C 180,E1 -6385.871,E2 -6385.871} C_VEL
LIN {X 0,Y 488.007,Z 380.117,A -85,B 0,C 180,E1 -6386.698,E2 -6386.698} C_VEL
LIN {X 0,Y 487.942,Z 381.525,A -85,B 0,C 180,E1 -6387.523,E2 -6387.523} C_VEL
LIN {X 0,Y 487.836,Z 383.144,A -85,B 0,C 180,E1 -6389.175,E2 -6389.175} C_VEL
LIN {X 0,Y 487.822,Z 383.381,A -85,B 0,C 180,E1 -6390,E2 -6390} C_VEL
LIN {X 0,Y 487.836,Z 383.196,A -85,B 0,C 180,E1 -6390.825,E2 -6390.825} C_VEL
LIN {X 0,Y 487.942,Z 381.645,A -85,B 0,C 180,E1 -6392.476,E2 -6392.476} C_VEL
LIN {X 0,Y 488.007,Z 380.288,A -85,B 0,C 180,E1 -6393.302,E2 -6393.302} C_VEL
LIN {X 0,Y 487.993,Z 377.424,A -85,B 0,C 180,E1 -6394.543,E2 -6394.543} C_VEL
LIN {X 0,Y 488.218,Z 372.443,A -85,B 0,C 180,E1 -6396.078,E2 -6396.078} C_VEL
LIN {X 0,Y 488.296,Z 366.552,A -85,B 0,C 180,E1 -6397.443,E2 -6397.443} C_VEL
LIN {X 0,Y 488.593,Z 359.763,A -85,B 0,C 180,E1 -6398.687,E2 -6398.687} C_VEL
LIN {X 0,Y 488.912,Z 351.289,A -85,B 0,C 180,E1 -6399.933,E2 -6399.933} C_VEL
LIN {X 0,Y 489.343,Z 342.569,A -85,B 0,C 180,E1 -6400.97,E2 -6400.97} C_VEL
LIN {X 0,Y 489.778,Z 331.831,A -85,B 0,C 180,E1 -6402.009,E2 -6402.009} C_VEL
LIN {X 0,Y 490.142,Z 320.431,A -85,B 0,C 180,E1 -6402.884,E2 -6402.884} C_VEL
LIN {X 0,Y 490.508,Z 308.989,A -85,B 0,C 180,E1 -6403.569,E2 -6403.569} C_VEL
LIN {X 0,Y 490.902,Z 296.34,A -85,B 0,C 180,E1 -6404.139,E2 -6404.139} C_VEL
LIN {X 0,Y 491.167,Z 283.85,A -85,B 0,C 180,E1 -6404.528,E2 -6404.528} C_VEL
LIN {X 0,Y 491.339,Z 267.903,A -85,B 0,C 180,E1 -6404.814,E2 -6404.814} C_VEL
LIN {X 0,Y 491.745,Z 185.319,A -85,B 0,C 180,E1 -6406.027,E2 -6406.027} C_VEL
LIN {X 0,Y 489.334,Z 172.376,A -85,B 0,C 180,E1 -6406.307,E2 -6406.307} C_VEL
LIN {X 0,Y 489.796,Z 155.851,A -85,B 0,C 180,E1 -6409.488,E2 -6409.488} C_VEL
LIN {X 0,Y 489.677,Z 150.336,A -85,B 0,C 180,E1 -6410.587,E2 -6410.587} C_VEL
LIN {X 0,Y 488.764,Z 145.104,A -85,B 0,C 180,E1 -6411.704,E2 -6411.704} C_VEL
LIN {X 0,Y 488.747,Z 145.106,A -85,B 0,C 180,E1 -6415.052,E2 -6415.052} C_VEL
LIN {X 0,Y 488.747,Z 145.101,A -85,B 0,C 180,E1 -6417.396,E2 -6417.396} C_VEL
LIN {X 0,Y 488.71,Z 145.109,A -85,B 0,C 180,E1 -6420.362,E2 -6420.362} C_VEL
LIN {X 0,Y 488.73,Z 145.102,A -85,B 0,C 180,E1 -6423.483,E2 -6423.483} C_VEL
LIN {X 0,Y 488.683,Z 145.115,A -85,B 0,C 180,E1 -6426.354,E2 -6426.354} C_VEL
LIN {X 0,Y 488.702,Z 145.106,A -85,B 0,C 180,E1 -6429.254,E2 -6429.254} C_VEL
LIN {X 0,Y 488.708,Z 145.106,A -85,B 0,C 180,E1 -6431.599,E2 -6431.599} C_VEL
LIN {X 0,Y 488.713,Z 145.105,A -85,B 0,C 180,E1 -6434.801,E2 -6434.801} C_VEL
LIN {X 0,Y 488.692,Z 145.108,A -85,B 0,C 180,E1 -6437.474,E2 -6437.474} C_VEL
LIN {X 0,Y 488.733,Z 145.105,A -85,B 0,C 180,E1 -6439.676,E2 -6439.676} C_VEL
LIN {X 0,Y 488.679,Z 145.108,A -85,B 0,C 180,E1 -6442.841,E2 -6442.841} C_VEL
LIN {X 0,Y 488.73,Z 145.11,A -85,B 0,C 180,E1 -6445.887,E2 -6445.887} C_VEL
LIN {X 0,Y 488.691,Z 145.107,A -85,B 0,C 180,E1 -6448.82,E2 -6448.82} C_VEL
LIN {X 0,Y 488.744,Z 145.109,A -85,B 0,C 180,E1 -6451.671,E2 -6451.671} C_VEL
LIN {X 0,Y 488.747,Z 145.1,A -85,B 0,C 180,E1 -6454.444,E2 -6454.444} C_VEL
LIN {X 0,Y 488.722,Z 145.107,A -85,B 0,C 180,E1 -6457.153,E2 -6457.153} C_VEL
LIN {X 0,Y 488.728,Z 145.106,A -85,B 0,C 180,E1 -6459.81,E2 -6459.81} C_VEL
LIN {X 0,Y 488.733,Z 145.102,A -85,B 0,C 180,E1 -6462.423,E2 -6462.423} C_VEL
LIN {X 0,Y 488.761,Z 145.103,A -85,B 0,C 180,E1 -6465,E2 -6465} C_VEL
LIN {X 0,Y 488.805,Z 145.093,A -85,B 0,C 180,E1 -6468.387,E2 -6468.387} C_VEL
LIN {X 0,Y 488.817,Z 145.092,A -85,B 0,C 180,E1 -6471.734,E2 -6471.734} C_VEL
LIN {X 0,Y 488.847,Z 145.088,A -85,B 0,C 180,E1 -6474.224,E2 -6474.224} C_VEL
LIN {X 0,Y 488.961,Z 145.074,A -85,B 0,C 180,E1 -6477.529,E2 -6477.529} C_VEL
LIN {X 0,Y 488.954,Z 145.082,A -85,B 0,C 180,E1 -6480.824,E2 -6480.824} C_VEL
LIN {X 0,Y 488.961,Z 145.078,A -85,B 0,C 180,E1 -6482.471,E2 -6482.471} C_VEL
LIN {X 0,Y 488.847,Z 145.088,A -85,B 0,C 180,E1 -6485.776,E2 -6485.776} C_VEL
LIN {X 0,Y 488.815,Z 145.096,A -85,B 0,C 180,E1 -6488.266,E2 -6488.266} C_VEL
LIN {X 0,Y 488.805,Z 145.093,A -85,B 0,C 180,E1 -6491.612,E2 -6491.612} C_VEL
LIN {X 0,Y 488.761,Z 145.099,A -85,B 0,C 180,E1 -6495,E2 -6495} C_VEL
LIN {X 0,Y 488.746,Z 145.106,A -85,B 0,C 180,E1 -6498.443,E2 -6498.443} C_VEL
LIN {X 0,Y 488.706,Z 145.105,A -85,B 0,C 180,E1 -6501.071,E2 -6501.071} C_VEL
LIN {X 0,Y 488.676,Z 145.113,A -85,B 0,C 180,E1 -6503.746,E2 -6503.746} C_VEL
LIN {X 0,Y 488.79,Z 145.095,A -85,B 0,C 180,E1 -6506.943,E2 -6506.943} C_VEL
LIN {X 0,Y 488.709,Z 145.107,A -85,B 0,C 180,E1 -6510.363,E2 -6510.363} C_VEL
LIN {X 0,Y 488.734,Z 145.106,A -85,B 0,C 180,E1 -6513.484,E2 -6513.484} C_VEL
LIN {X 0,Y 488.672,Z 145.11,A -85,B 0,C 180,E1 -6516.353,E2 -6516.353} C_VEL
LIN {X 0,Y 488.7,Z 145.109,A -85,B 0,C 180,E1 -6519.255,E2 -6519.255} C_VEL
LIN {X 0,Y 488.688,Z 145.107,A -85,B 0,C 180,E1 -6522.526,E2 -6522.526} C_VEL
LIN {X 0,Y 488.701,Z 145.111,A -85,B 0,C 180,E1 -6525.198,E2 -6525.198} C_VEL
LIN {X 0,Y 488.679,Z 145.109,A -85,B 0,C 180,E1 -6528.582,E2 -6528.582} C_VEL
LIN {X 0,Y 488.677,Z 145.11,A -85,B 0,C 180,E1 -6531.8,E2 -6531.8} C_VEL
LIN {X 0,Y 488.72,Z 145.111,A -85,B 0,C 180,E1 -6535.053,E2 -6535.053} C_VEL
LIN {X 0,Y 488.701,Z 145.106,A -85,B 0,C 180,E1 -6538.047,E2 -6538.047} C_VEL
LIN {X 0,Y 488.701,Z 145.113,A -85,B 0,C 180,E1 -6540.728,E2 -6540.728} C_VEL
LIN {X 0,Y 488.686,Z 145.111,A -85,B 0,C 180,E1 -6543.524,E2 -6543.524} C_VEL
LIN {X 0,Y 488.727,Z 145.214,A -85,B 0,C 180,E1 -6545.255,E2 -6545.255} C_VEL
LIN {X 0,Y 490.418,Z 154.071,A -85,B 0,C 180,E1 -6546.924,E2 -6546.924} C_VEL
LIN {X 0,Y 490.303,Z 163.101,A -85,B 0,C 180,E1 -6548.518,E2 -6548.518} C_VEL
LIN {X 0,Y 489.607,Z 182.092,A -85,B 0,C 180,E1 -6551.808,E2 -6551.808} C_VEL
LIN {X 0,Y 489.269,Z 193.534,A -85,B 0,C 180,E1 -6553.735,E2 -6553.735} C_VEL
LIN {X 0,Y 491.688,Z 208.751,A -85,B 0,C 180,E1 -6554.043,E2 -6554.043} C_VEL
LIN {X 0,Y 491.118,Z 301.348,A -85,B 0,C 180,E1 -6555.418,E2 -6555.418} C_VEL
LIN {X 0,Y 490.826,Z 314.622,A -85,B 0,C 180,E1 -6555.78,E2 -6555.78} C_VEL
LIN {X 0,Y 490.459,Z 326.784,A -85,B 0,C 180,E1 -6556.271,E2 -6556.271} C_VEL
LIN {X 0,Y 490.035,Z 339.059,A -85,B 0,C 180,E1 -6556.945,E2 -6556.945} C_VEL
LIN {X 0,Y 489.624,Z 350.652,A -85,B 0,C 180,E1 -6557.777,E2 -6557.777} C_VEL
LIN {X 0,Y 489.255,Z 361.092,A -85,B 0,C 180,E1 -6558.713,E2 -6558.713} C_VEL
LIN {X 0,Y 488.835,Z 369.625,A -85,B 0,C 180,E1 -6559.647,E2 -6559.647} C_VEL
LIN {X 0,Y 488.544,Z 377.5,A -85,B 0,C 180,E1 -6560.686,E2 -6560.686} C_VEL
LIN {X 0,Y 488.271,Z 385.191,A -85,B 0,C 180,E1 -6561.933,E2 -6561.933} C_VEL
LIN {X 0,Y 488.096,Z 392.282,A -85,B 0,C 180,E1 -6563.385,E2 -6563.385} C_VEL
LIN {X 0,Y 488.021,Z 396.999,A -85,B 0,C 180,E1 -6564.629,E2 -6564.629} C_VEL
LIN {X 0,Y 487.926,Z 400.601,A -85,B 0,C 180,E1 -6565.87,E2 -6565.87} C_VEL
LIN {X 0,Y 487.964,Z 402.461,A -85,B 0,C 180,E1 -6566.697,E2 -6566.697} C_VEL
LIN {X 0,Y 487.891,Z 404.848,A -85,B 0,C 180,E1 -6568.349,E2 -6568.349} C_VEL
LIN {X 0,Y 487.821,Z 405.67,A -85,B 0,C 180,E1 -6570,E2 -6570} C_VEL
LIN {X 0,Y 487.891,Z 404.85,A -85,B 0,C 180,E1 -6571.651,E2 -6571.651} C_VEL
LIN {X 0,Y 487.964,Z 402.464,A -85,B 0,C 180,E1 -6573.303,E2 -6573.303} C_VEL
LIN {X 0,Y 487.919,Z 399.532,A -85,B 0,C 180,E1 -6574.544,E2 -6574.544} C_VEL
LIN {X 0,Y 488.02,Z 395.565,A -85,B 0,C 180,E1 -6575.786,E2 -6575.786} C_VEL
LIN {X 0,Y 488.178,Z 389.463,A -85,B 0,C 180,E1 -6577.237,E2 -6577.237} C_VEL
LIN {X 0,Y 488.353,Z 382.793,A -85,B 0,C 180,E1 -6578.483,E2 -6578.483} C_VEL
LIN {X 0,Y 488.694,Z 374.518,A -85,B 0,C 180,E1 -6579.728,E2 -6579.728} C_VEL
LIN {X 0,Y 488.994,Z 366.035,A -85,B 0,C 180,E1 -6580.768,E2 -6580.768} C_VEL
LIN {X 0,Y 489.485,Z 355.556,A -85,B 0,C 180,E1 -6581.806,E2 -6581.806} C_VEL
LIN {X 0,Y 489.833,Z 343.818,A -85,B 0,C 180,E1 -6582.739,E2 -6582.739} C_VEL
LIN {X 0,Y 490.283,Z 331.892,A -85,B 0,C 180,E1 -6583.47,E2 -6583.47} C_VEL
LIN {X 0,Y 490.675,Z 319.549,A -85,B 0,C 180,E1 -6584.04,E2 -6584.04} C_VEL
LIN {X 0,Y 491.047,Z 306.883,A -85,B 0,C 180,E1 -6584.452,E2 -6584.452} C_VEL
LIN {X 0,Y 491.206,Z 293.654,A -85,B 0,C 180,E1 -6584.712,E2 -6584.712} C_VEL
LIN {X 0,Y 491.606,Z 208.037,A -85,B 0,C 180,E1 -6585.969,E2 -6585.969} C_VEL
LIN {X 0,Y 489.263,Z 193.158,A -85,B 0,C 180,E1 -6586.294,E2 -6586.294} C_VEL
LIN {X 0,Y 489.864,Z 174.587,A -85,B 0,C 180,E1 -6589.485,E2 -6589.485} C_VEL
LIN {X 0,Y 490.384,Z 159.574,A -85,B 0,C 180,E1 -6592.099,E2 -6592.099} C_VEL
LIN {X 0,Y 490.43,Z 154.045,A -85,B 0,C 180,E1 -6593.077,E2 -6593.077} C_VEL
LIN {X 0,Y 488.707,Z 145.113,A -85,B 0,C 180,E1 -6594.795,E2 -6594.795} C_VEL
LIN {X 0,Y 488.687,Z 145.111,A -85,B 0,C 180,E1 -6597.4,E2 -6597.4} C_VEL
LIN {X 0,Y 488.702,Z 145.105,A -85,B 0,C 180,E1 -6600.361,E2 -6600.361} C_VEL
LIN {X 0,Y 488.711,Z 145.106,A -85,B 0,C 180,E1 -6603.48,E2 -6603.48} C_VEL
LIN {X 0,Y 488.683,Z 145.11,A -85,B 0,C 180,E1 -6606.354,E2 -6606.354} C_VEL
LIN {X 0,Y 488.694,Z 145.109,A -85,B 0,C 180,E1 -6609.255,E2 -6609.255} C_VEL
LIN {X 0,Y 488.687,Z 145.114,A -85,B 0,C 180,E1 -6612.526,E2 -6612.526} C_VEL
LIN {X 0,Y 488.701,Z 145.107,A -85,B 0,C 180,E1 -6615.197,E2 -6615.197} C_VEL
LIN {X 0,Y 488.694,Z 145.113,A -85,B 0,C 180,E1 -6618.583,E2 -6618.583} C_VEL
LIN {X 0,Y 488.703,Z 145.107,A -85,B 0,C 180,E1 -6620.947,E2 -6620.947} C_VEL
LIN {X 0,Y 488.669,Z 145.112,A -85,B 0,C 180,E1 -6623.867,E2 -6623.867} C_VEL
LIN {X 0,Y 488.738,Z 145.102,A -85,B 0,C 180,E1 -6626.877,E2 -6626.877} C_VEL
LIN {X 0,Y 488.722,Z 145.107,A -85,B 0,C 180,E1 -6629.78,E2 -6629.78} C_VEL
LIN {X 0,Y 488.725,Z 145.103,A -85,B 0,C 180,E1 -6633.072,E2 -6633.072} C_VEL
LIN {X 0,Y 488.71,Z 145.106,A -85,B 0,C 180,E1 -6635.352,E2 -6635.352} C_VEL
LIN {X 0,Y 488.697,Z 145.112,A -85,B 0,C 180,E1 -6638.043,E2 -6638.043} C_VEL
LIN {X 0,Y 488.741,Z 145.101,A -85,B 0,C 180,E1 -6640.687,E2 -6640.687} C_VEL
LIN {X 0,Y 488.76,Z 145.101,A -85,B 0,C 180,E1 -6644.145,E2 -6644.145} C_VEL
LIN {X 0,Y 488.73,Z 145.102,A -85,B 0,C 180,E1 -6646.698,E2 -6646.698} C_VEL
LIN {X 0,Y 488.736,Z 145.105,A -85,B 0,C 180,E1 -6649.226,E2 -6649.226} C_VEL
LIN {X 0,Y 488.862,Z 145.086,A -85,B 0,C 180,E1 -6652.566,E2 -6652.566} C_VEL
LIN {X 0,Y 488.81,Z 145.096,A -85,B 0,C 180,E1 -6655.051,E2 -6655.051} C_VEL
LIN {X 0,Y 488.961,Z 145.078,A -85,B 0,C 180,E1 -6657.529,E2 -6657.529} C_VEL
LIN {X 0,Y 488.969,Z 145.073,A -85,B 0,C 180,E1 -6660,E2 -6660} C_VEL
LIN {X 0,Y 488.961,Z 145.074,A -85,B 0,C 180,E1 -6662.471,E2 -6662.471} C_VEL
LIN {X 0,Y 488.842,Z 145.089,A -85,B 0,C 180,E1 -6665.776,E2 -6665.776} C_VEL
LIN {X 0,Y 488.816,Z 145.092,A -85,B 0,C 180,E1 -6668.266,E2 -6668.266} C_VEL
LIN {X 0,Y 488.805,Z 145.093,A -85,B 0,C 180,E1 -6671.613,E2 -6671.613} C_VEL
LIN {X 0,Y 488.762,Z 145.103,A -85,B 0,C 180,E1 -6675,E2 -6675} C_VEL
LIN {X 0,Y 488.755,Z 145.104,A -85,B 0,C 180,E1 -6678.442,E2 -6678.442} C_VEL
LIN {X 0,Y 488.707,Z 145.107,A -85,B 0,C 180,E1 -6681.071,E2 -6681.071} C_VEL
LIN {X 0,Y 488.689,Z 145.107,A -85,B 0,C 180,E1 -6683.746,E2 -6683.746} C_VEL
LIN {X 0,Y 488.792,Z 145.096,A -85,B 0,C 180,E1 -6686.944,E2 -6686.944} C_VEL
LIN {X 0,Y 488.71,Z 145.113,A -85,B 0,C 180,E1 -6690.363,E2 -6690.363} C_VEL
LIN {X 0,Y 488.735,Z 145.102,A -85,B 0,C 180,E1 -6693.484,E2 -6693.484} C_VEL
LIN {X 0,Y 488.683,Z 145.113,A -85,B 0,C 180,E1 -6696.355,E2 -6696.355} C_VEL
LIN {X 0,Y 488.702,Z 145.106,A -85,B 0,C 180,E1 -6699.254,E2 -6699.254} C_VEL
LIN {X 0,Y 488.709,Z 145.108,A -85,B 0,C 180,E1 -6701.6,E2 -6701.6} C_VEL
LIN {X 0,Y 488.713,Z 145.104,A -85,B 0,C 180,E1 -6704.802,E2 -6704.802} C_VEL
LIN {X 0,Y 488.693,Z 145.11,A -85,B 0,C 180,E1 -6707.475,E2 -6707.475} C_VEL
LIN {X 0,Y 488.734,Z 145.109,A -85,B 0,C 180,E1 -6709.677,E2 -6709.677} C_VEL
LIN {X 0,Y 488.681,Z 145.108,A -85,B 0,C 180,E1 -6712.841,E2 -6712.841} C_VEL
LIN {X 0,Y 488.725,Z 145.107,A -85,B 0,C 180,E1 -6715.887,E2 -6715.887} C_VEL
LIN {X 0,Y 488.693,Z 145.108,A -85,B 0,C 180,E1 -6718.82,E2 -6718.82} C_VEL
LIN {X 0,Y 488.746,Z 145.106,A -85,B 0,C 180,E1 -6721.671,E2 -6721.671} C_VEL
LIN {X 0,Y 488.744,Z 145.102,A -85,B 0,C 180,E1 -6724.331,E2 -6724.331} C_VEL
LIN {X 0,Y 488.089,Z 145.188,A -85,B 0,C 180,E1 -6725.019,E2 -6725.019} C_VEL
LIN {X 0,Y 485.195,Z 145.548,A -85,B 0,C 180,E1 -6726.135,E2 -6726.135} C_VEL
LIN {X 0,Y 482.758,Z 145.852,A -85,B 0,C 180,E1 -6727.035,E2 -6727.035} C_VEL
LIN {X 0,Y 481.745,Z 145.978,A -85,B 0,C 180,E1 -6727.73,E2 -6727.73} C_VEL
LIN {X 0,Y 481.681,Z 145.985,A -85,B 0,C 180,E1 -6727.966,E2 -6727.966} C_VEL
LIN {X 0,Y 481.702,Z 146.101,A -85,B 0,C 180,E1 -6728.271,E2 -6728.271} C_VEL
LIN {X 0,Y 482.891,Z 153.265,A -85,B 0,C 180,E1 -6729.778,E2 -6729.778} C_VEL
LIN {X 0,Y 482.542,Z 166.628,A -85,B 0,C 180,E1 -6732.409,E2 -6732.409} C_VEL
LIN {X 0,Y 482.398,Z 172.591,A -85,B 0,C 180,E1 -6733.549,E2 -6733.549} C_VEL
LIN {X 0,Y 485,Z 186.777,A -85,B 0,C 180,E1 -6733.855,E2 -6733.855} C_VEL
LIN {X 0,Y 484.371,Z 280.107,A -85,B 0,C 180,E1 -6735.264,E2 -6735.264} C_VEL
LIN {X 0,Y 484.048,Z 294.006,A -85,B 0,C 180,E1 -6735.657,E2 -6735.657} C_VEL
LIN {X 0,Y 483.706,Z 306.434,A -85,B 0,C 180,E1 -6736.183,E2 -6736.183} C_VEL
LIN {X 0,Y 483.359,Z 317.87,A -85,B 0,C 180,E1 -6736.839,E2 -6736.839} C_VEL
LIN {X 0,Y 482.973,Z 328.391,A -85,B 0,C 180,E1 -6737.606,E2 -6737.606} C_VEL
LIN {X 0,Y 482.519,Z 338.868,A -85,B 0,C 180,E1 -6738.554,E2 -6738.554} C_VEL
LIN {X 0,Y 482.142,Z 347.429,A -85,B 0,C 180,E1 -6739.502,E2 -6739.502} C_VEL
LIN {X 0,Y 481.745,Z 355.314,A -85,B 0,C 180,E1 -6740.554,E2 -6740.554} C_VEL
LIN {X 0,Y 481.417,Z 363.023,A -85,B 0,C 180,E1 -6741.817,E2 -6741.817} C_VEL
LIN {X 0,Y 481.162,Z 370.094,A -85,B 0,C 180,E1 -6743.29,E2 -6743.29} C_VEL
LIN {X 0,Y 481.027,Z 374.807,A -85,B 0,C 180,E1 -6744.551,E2 -6744.551} C_VEL
LIN {X 0,Y 480.945,Z 378.415,A -85,B 0,C 180,E1 -6745.81,E2 -6745.81} C_VEL
LIN {X 0,Y 480.933,Z 380.28,A -85,B 0,C 180,E1 -6746.649,E2 -6746.649} C_VEL
LIN {X 0,Y 480.855,Z 381.688,A -85,B 0,C 180,E1 -6747.487,E2 -6747.487} C_VEL
LIN {X 0,Y 480.824,Z 382.688,A -85,B 0,C 180,E1 -6748.325,E2 -6748.325} C_VEL
LIN {X 0,Y 480.746,Z 383.542,A -85,B 0,C 180,E1 -6750,E2 -6750} C_VEL
LIN {X 0,Y 480.762,Z 383.357,A -85,B 0,C 180,E1 -6750.838,E2 -6750.838} C_VEL
LIN {X 0,Y 480.825,Z 382.772,A -85,B 0,C 180,E1 -6751.675,E2 -6751.675} C_VEL
LIN {X 0,Y 480.933,Z 380.449,A -85,B 0,C 180,E1 -6753.351,E2 -6753.351} C_VEL
LIN {X 0,Y 480.899,Z 377.586,A -85,B 0,C 180,E1 -6754.61,E2 -6754.61} C_VEL
LIN {X 0,Y 481.12,Z 373.696,A -85,B 0,C 180,E1 -6755.869,E2 -6755.869} C_VEL
LIN {X 0,Y 481.196,Z 368.684,A -85,B 0,C 180,E1 -6757.131,E2 -6757.131} C_VEL
LIN {X 0,Y 481.457,Z 362.373,A -85,B 0,C 180,E1 -6758.394,E2 -6758.394} C_VEL
LIN {X 0,Y 481.79,Z 354.471,A -85,B 0,C 180,E1 -6759.657,E2 -6759.657} C_VEL
LIN {X 0,Y 482.134,Z 346.417,A -85,B 0,C 180,E1 -6760.711,E2 -6760.711} C_VEL
LIN {X 0,Y 482.608,Z 336.586,A -85,B 0,C 180,E1 -6761.764,E2 -6761.764} C_VEL
LIN {X 0,Y 483.054,Z 325.568,A -85,B 0,C 180,E1 -6762.71,E2 -6762.71} C_VEL
LIN {X 0,Y 483.433,Z 314.706,A -85,B 0,C 180,E1 -6763.45,E2 -6763.45} C_VEL
LIN {X 0,Y 483.828,Z 302.746,A -85,B 0,C 180,E1 -6764.082,E2 -6764.082} C_VEL
LIN {X 0,Y 484.197,Z 289.644,A -85,B 0,C 180,E1 -6764.58,E2 -6764.58} C_VEL
LIN {X 0,Y 484.374,Z 276.487,A -85,B 0,C 180,E1 -6764.897,E2 -6764.897} C_VEL
LIN {X 0,Y 484.935,Z 186.319,A -85,B 0,C 180,E1 -6766.246,E2 -6766.246} C_VEL
LIN {X 0,Y 482.392,Z 172.521,A -85,B 0,C 180,E1 -6766.548,E2 -6766.548} C_VEL
LIN {X 0,Y 482.874,Z 155.942,A -85,B 0,C 180,E1 -6769.779,E2 -6769.779} C_VEL
LIN {X 0,Y 482.595,Z 150.919,A -85,B 0,C 180,E1 -6770.801,E2 -6770.801} C_VEL
LIN {X 0,Y 481.697,Z 145.984,A -85,B 0,C 180,E1 -6771.87,E2 -6771.87} C_VEL
LIN {X 0,Y 481.713,Z 145.981,A -85,B 0,C 180,E1 -6775.236,E2 -6775.236} C_VEL
LIN {X 0,Y 481.701,Z 145.978,A -85,B 0,C 180,E1 -6777.832,E2 -6777.832} C_VEL
LIN {X 0,Y 481.646,Z 145.992,A -85,B 0,C 180,E1 -6780.711,E2 -6780.711} C_VEL
LIN {X 0,Y 481.676,Z 145.981,A -85,B 0,C 180,E1 -6783.729,E2 -6783.729} C_VEL
LIN {X 0,Y 481.627,Z 145.991,A -85,B 0,C 180,E1 -6786.747,E2 -6786.747} C_VEL
LIN {X 0,Y 481.678,Z 145.984,A -85,B 0,C 180,E1 -6789.94,E2 -6789.94} C_VEL
LIN {X 0,Y 481.64,Z 145.985,A -85,B 0,C 180,E1 -6793.299,E2 -6793.299} C_VEL
LIN {X 0,Y 481.659,Z 145.985,A -85,B 0,C 180,E1 -6795.64,E2 -6795.64} C_VEL
LIN {X 0,Y 481.657,Z 145.983,A -85,B 0,C 180,E1 -6798.958,E2 -6798.958} C_VEL
LIN {X 0,Y 481.655,Z 145.992,A -85,B 0,C 180,E1 -6801.992,E2 -6801.992} C_VEL
LIN {X 0,Y 481.688,Z 145.981,A -85,B 0,C 180,E1 -6805.318,E2 -6805.318} C_VEL
LIN {X 0,Y 481.644,Z 145.987,A -85,B 0,C 180,E1 -6808.311,E2 -6808.311} C_VEL
LIN {X 0,Y 481.699,Z 145.98,A -85,B 0,C 180,E1 -6811.218,E2 -6811.218} C_VEL
LIN {X 0,Y 481.701,Z 145.98,A -85,B 0,C 180,E1 -6814.043,E2 -6814.043} C_VEL
LIN {X 0,Y 481.674,Z 145.982,A -85,B 0,C 180,E1 -6816.812,E2 -6816.812} C_VEL
LIN {X 0,Y 481.697,Z 145.986,A -85,B 0,C 180,E1 -6819.503,E2 -6819.503} C_VEL
LIN {X 0,Y 481.707,Z 145.977,A -85,B 0,C 180,E1 -6822.158,E2 -6822.158} C_VEL
LIN {X 0,Y 481.742,Z 145.975,A -85,B 0,C 180,E1 -6824.776,E2 -6824.776} C_VEL
LIN {X 0,Y 481.75,Z 145.971,A -85,B 0,C 180,E1 -6828.215,E2 -6828.215} C_VEL
LIN {X 0,Y 481.762,Z 145.972,A -85,B 0,C 180,E1 -6831.612,E2 -6831.612} C_VEL
LIN {X 0,Y 481.807,Z 145.965,A -85,B 0,C 180,E1 -6834.139,E2 -6834.139} C_VEL
LIN {X 0,Y 481.928,Z 145.951,A -85,B 0,C 180,E1 -6837.492,E2 -6837.492} C_VEL
LIN {X 0,Y 481.905,Z 145.96,A -85,B 0,C 180,E1 -6840.836,E2 -6840.836} C_VEL
LIN {X 0,Y 481.927,Z 145.954,A -85,B 0,C 180,E1 -6842.507,E2 -6842.507} C_VEL
LIN {X 0,Y 481.808,Z 145.965,A -85,B 0,C 180,E1 -6845.861,E2 -6845.861} C_VEL
LIN {X 0,Y 481.76,Z 145.976,A -85,B 0,C 180,E1 -6848.388,E2 -6848.388} C_VEL
LIN {X 0,Y 481.75,Z 145.972,A -85,B 0,C 180,E1 -6851.785,E2 -6851.785} C_VEL
LIN {X 0,Y 481.742,Z 145.973,A -85,B 0,C 180,E1 -6855.224,E2 -6855.224} C_VEL
LIN {X 0,Y 481.707,Z 145.979,A -85,B 0,C 180,E1 -6858.722,E2 -6858.722} C_VEL
LIN {X 0,Y 481.644,Z 145.985,A -85,B 0,C 180,E1 -6861.395,E2 -6861.395} C_VEL
LIN {X 0,Y 481.657,Z 145.991,A -85,B 0,C 180,E1 -6864.114,E2 -6864.114} C_VEL
LIN {X 0,Y 481.744,Z 145.972,A -85,B 0,C 180,E1 -6867.139,E2 -6867.139} C_VEL
LIN {X 0,Y 481.677,Z 145.987,A -85,B 0,C 180,E1 -6869.741,E2 -6869.741} C_VEL
LIN {X 0,Y 481.671,Z 145.982,A -85,B 0,C 180,E1 -6872.674,E2 -6872.674} C_VEL
LIN {X 0,Y 481.66,Z 145.985,A -85,B 0,C 180,E1 -6875.204,E2 -6875.204} C_VEL
LIN {X 0,Y 481.669,Z 145.982,A -85,B 0,C 180,E1 -6878.859,E2 -6878.859} C_VEL
LIN {X 0,Y 481.646,Z 145.988,A -85,B 0,C 180,E1 -6881.912,E2 -6881.912} C_VEL
LIN {X 0,Y 481.654,Z 145.984,A -85,B 0,C 180,E1 -6884.458,E2 -6884.458} C_VEL
LIN {X 0,Y 481.639,Z 145.988,A -85,B 0,C 180,E1 -6887.839,E2 -6887.839} C_VEL
LIN {X 0,Y 481.666,Z 145.989,A -85,B 0,C 180,E1 -6891.141,E2 -6891.141} C_VEL
LIN {X 0,Y 481.636,Z 145.986,A -85,B 0,C 180,E1 -6894.291,E2 -6894.291} C_VEL
LIN {X 0,Y 481.67,Z 145.986,A -85,B 0,C 180,E1 -6897.326,E2 -6897.326} C_VEL
LIN {X 0,Y 481.666,Z 145.986,A -85,B 0,C 180,E1 -6900.258,E2 -6900.258} C_VEL
LIN {X 0,Y 481.662,Z 145.988,A -85,B 0,C 180,E1 -6903.107,E2 -6903.107} C_VEL
LIN {X 0,Y 481.667,Z 146.065,A -85,B 0,C 180,E1 -6905.054,E2 -6905.054} C_VEL
LIN {X 0,Y 483.511,Z 155.669,A -85,B 0,C 180,E1 -6906.893,E2 -6906.893} C_VEL
LIN {X 0,Y 483.202,Z 166.936,A -85,B 0,C 180,E1 -6908.901,E2 -6908.901} C_VEL
LIN {X 0,Y 482.557,Z 184.428,A -85,B 0,C 180,E1 -6911.972,E2 -6911.972} C_VEL
LIN {X 0,Y 482.276,Z 193.24,A -85,B 0,C 180,E1 -6913.49,E2 -6913.49} C_VEL
LIN {X 0,Y 484.872,Z 210.16,A -85,B 0,C 180,E1 -6913.836,E2 -6913.836} C_VEL
LIN {X 0,Y 484.256,Z 301.195,A -85,B 0,C 180,E1 -6915.206,E2 -6915.206} C_VEL
LIN {X 0,Y 483.948,Z 314.466,A -85,B 0,C 180,E1 -6915.573,E2 -6915.573} C_VEL
LIN {X 0,Y 483.582,Z 326.627,A -85,B 0,C 180,E1 -6916.072,E2 -6916.072} C_VEL
LIN {X 0,Y 483.155,Z 337.385,A -85,B 0,C 180,E1 -6916.66,E2 -6916.66} C_VEL
LIN {X 0,Y 482.706,Z 348.828,A -85,B 0,C 180,E1 -6917.462,E2 -6917.462} C_VEL
LIN {X 0,Y 482.266,Z 359.858,A -85,B 0,C 180,E1 -6918.441,E2 -6918.441} C_VEL
LIN {X 0,Y 481.819,Z 369.464,A -85,B 0,C 180,E1 -6919.495,E2 -6919.495} C_VEL
LIN {X 0,Y 481.493,Z 377.339,A -85,B 0,C 180,E1 -6920.549,E2 -6920.549} C_VEL
LIN {X 0,Y 481.222,Z 385.029,A -85,B 0,C 180,E1 -6921.814,E2 -6921.814} C_VEL
LIN {X 0,Y 481.012,Z 392.119,A -85,B 0,C 180,E1 -6923.288,E2 -6923.288} C_VEL
LIN {X 0,Y 480.933,Z 396.837,A -85,B 0,C 180,E1 -6924.55,E2 -6924.55} C_VEL
LIN {X 0,Y 480.826,Z 400.439,A -85,B 0,C 180,E1 -6925.809,E2 -6925.809} C_VEL
LIN {X 0,Y 480.87,Z 402.299,A -85,B 0,C 180,E1 -6926.649,E2 -6926.649} C_VEL
LIN {X 0,Y 480.823,Z 403.692,A -85,B 0,C 180,E1 -6927.487,E2 -6927.487} C_VEL
LIN {X 0,Y 480.761,Z 405.293,A -85,B 0,C 180,E1 -6929.162,E2 -6929.162} C_VEL
LIN {X 0,Y 480.745,Z 405.508,A -85,B 0,C 180,E1 -6930,E2 -6930} C_VEL
LIN {X 0,Y 480.792,Z 404.687,A -85,B 0,C 180,E1 -6931.675,E2 -6931.675} C_VEL
LIN {X 0,Y 480.823,Z 403.694,A -85,B 0,C 180,E1 -6932.513,E2 -6932.513} C_VEL
LIN {X 0,Y 480.87,Z 402.302,A -85,B 0,C 180,E1 -6933.351,E2 -6933.351} C_VEL
LIN {X 0,Y 480.837,Z 399.369,A -85,B 0,C 180,E1 -6934.611,E2 -6934.611} C_VEL
LIN {X 0,Y 480.924,Z 395.401,A -85,B 0,C 180,E1 -6935.871,E2 -6935.871} C_VEL
LIN {X 0,Y 481.081,Z 390.296,A -85,B 0,C 180,E1 -6937.133,E2 -6937.133} C_VEL
LIN {X 0,Y 481.264,Z 383.865,A -85,B 0,C 180,E1 -6938.397,E2 -6938.397} C_VEL
LIN {X 0,Y 481.585,Z 375.844,A -85,B 0,C 180,E1 -6939.661,E2 -6939.661} C_VEL
LIN {X 0,Y 481.883,Z 367.669,A -85,B 0,C 180,E1 -6940.717,E2 -6940.717} C_VEL
LIN {X 0,Y 482.374,Z 357.702,A -85,B 0,C 180,E1 -6941.769,E2 -6941.769} C_VEL
LIN {X 0,Y 482.718,Z 347.869,A -85,B 0,C 180,E1 -6942.614,E2 -6942.614} C_VEL
LIN {X 0,Y 483.153,Z 337.19,A -85,B 0,C 180,E1 -6943.351,E2 -6943.351} C_VEL
LIN {X 0,Y 483.63,Z 324.328,A -85,B 0,C 180,E1 -6944.034,E2 -6944.034} C_VEL
LIN {X 0,Y 483.989,Z 312.127,A -85,B 0,C 180,E1 -6944.506,E2 -6944.506} C_VEL
LIN {X 0,Y 484.31,Z 299.786,A -85,B 0,C 180,E1 -6944.819,E2 -6944.819} C_VEL
LIN {X 0,Y 484.812,Z 209.069,A -85,B 0,C 180,E1 -6946.181,E2 -6946.181} C_VEL
LIN {X 0,Y 482.264,Z 193.148,A -85,B 0,C 180,E1 -6946.51,E2 -6946.51} C_VEL
LIN {X 0,Y 482.881,Z 175.674,A -85,B 0,C 180,E1 -6949.557,E2 -6949.557} C_VEL
LIN {X 0,Y 483.45,Z 160.665,A -85,B 0,C 180,E1 -6952.208,E2 -6952.208} C_VEL
LIN {X 0,Y 483.51,Z 155.652,A -85,B 0,C 180,E1 -6953.107,E2 -6953.107} C_VEL
LIN {X 0,Y 481.656,Z 145.992,A -85,B 0,C 180,E1 -6954.976,E2 -6954.976} C_VEL
LIN {X 0,Y 481.652,Z 145.984,A -85,B 0,C 180,E1 -6957.835,E2 -6957.835} C_VEL
LIN {X 0,Y 481.639,Z 145.989,A -85,B 0,C 180,E1 -6960.711,E2 -6960.711} C_VEL
LIN {X 0,Y 481.676,Z 145.981,A -85,B 0,C 180,E1 -6963.729,E2 -6963.729} C_VEL
LIN {X 0,Y 481.626,Z 145.994,A -85,B 0,C 180,E1 -6966.747,E2 -6966.747} C_VEL
LIN {X 0,Y 481.657,Z 145.983,A -85,B 0,C 180,E1 -6969.942,E2 -6969.942} C_VEL
LIN {X 0,Y 481.626,Z 145.989,A -85,B 0,C 180,E1 -6973.146,E2 -6973.146} C_VEL
LIN {X 0,Y 481.653,Z 145.984,A -85,B 0,C 180,E1 -6975.641,E2 -6975.641} C_VEL
LIN {X 0,Y 481.649,Z 145.986,A -85,B 0,C 180,E1 -6978.957,E2 -6978.957} C_VEL
LIN {X 0,Y 481.65,Z 145.987,A -85,B 0,C 180,E1 -6981.993,E2 -6981.993} C_VEL
LIN {X 0,Y 481.687,Z 145.979,A -85,B 0,C 180,E1 -6985.318,E2 -6985.318} C_VEL
LIN {X 0,Y 481.644,Z 145.991,A -85,B 0,C 180,E1 -6988.311,E2 -6988.311} C_VEL
LIN {X 0,Y 481.674,Z 145.981,A -85,B 0,C 180,E1 -6991.217,E2 -6991.217} C_VEL
LIN {X 0,Y 481.669,Z 145.99,A -85,B 0,C 180,E1 -6994.041,E2 -6994.041} C_VEL
LIN {X 0,Y 481.674,Z 145.981,A -85,B 0,C 180,E1 -6996.812,E2 -6996.812} C_VEL
LIN {X 0,Y 481.695,Z 145.982,A -85,B 0,C 180,E1 -6999.503,E2 -6999.503} C_VEL
LIN {X 0,Y 481.691,Z 145.982,A -85,B 0,C 180,E1 -7002.158,E2 -7002.158} C_VEL
LIN {X 0,Y 481.742,Z 145.973,A -85,B 0,C 180,E1 -7004.776,E2 -7004.776} C_VEL
LIN {X 0,Y 481.75,Z 145.973,A -85,B 0,C 180,E1 -7008.215,E2 -7008.215} C_VEL
LIN {X 0,Y 481.761,Z 145.977,A -85,B 0,C 180,E1 -7011.612,E2 -7011.612} C_VEL
LIN {X 0,Y 481.808,Z 145.965,A -85,B 0,C 180,E1 -7014.14,E2 -7014.14} C_VEL
LIN {X 0,Y 481.928,Z 145.955,A -85,B 0,C 180,E1 -7017.493,E2 -7017.493} C_VEL
LIN {X 0,Y 481.94,Z 145.948,A -85,B 0,C 180,E1 -7020,E2 -7020} C_VEL
LIN {X 0,Y 481.928,Z 145.95,A -85,B 0,C 180,E1 -7022.508,E2 -7022.508} C_VEL
LIN {X 0,Y 481.801,Z 145.965,A -85,B 0,C 180,E1 -7025.861,E2 -7025.861} C_VEL
LIN {X 0,Y 481.761,Z 145.972,A -85,B 0,C 180,E1 -7028.388,E2 -7028.388} C_VEL
LIN {X 0,Y 481.751,Z 145.971,A -85,B 0,C 180,E1 -7031.785,E2 -7031.785} C_VEL
LIN {X 0,Y 481.743,Z 145.975,A -85,B 0,C 180,E1 -7035.224,E2 -7035.224} C_VEL
LIN {X 0,Y 481.713,Z 145.984,A -85,B 0,C 180,E1 -7038.722,E2 -7038.722} C_VEL
LIN {X 0,Y 481.645,Z 145.985,A -85,B 0,C 180,E1 -7041.395,E2 -7041.395} C_VEL
LIN {X 0,Y 481.674,Z 145.984,A -85,B 0,C 180,E1 -7044.113,E2 -7044.113} C_VEL
LIN {X 0,Y 481.747,Z 145.973,A -85,B 0,C 180,E1 -7047.139,E2 -7047.139} C_VEL
LIN {X 0,Y 481.679,Z 145.982,A -85,B 0,C 180,E1 -7049.741,E2 -7049.741} C_VEL
LIN {X 0,Y 481.672,Z 145.984,A -85,B 0,C 180,E1 -7052.674,E2 -7052.674} C_VEL
LIN {X 0,Y 481.637,Z 145.988,A -85,B 0,C 180,E1 -7055.71,E2 -7055.71} C_VEL
LIN {X 0,Y 481.672,Z 145.982,A -85,B 0,C 180,E1 -7058.859,E2 -7058.859} C_VEL
LIN {X 0,Y 481.654,Z 145.991,A -85,B 0,C 180,E1 -7061.913,E2 -7061.913} C_VEL
LIN {X 0,Y 481.661,Z 145.984,A -85,B 0,C 180,E1 -7064.458,E2 -7064.458} C_VEL
LIN {X 0,Y 481.649,Z 145.992,A -85,B 0,C 180,E1 -7067.84,E2 -7067.84} C_VEL
LIN {X 0,Y 481.662,Z 145.982,A -85,B 0,C 180,E1 -7070.654,E2 -7070.654} C_VEL
LIN {X 0,Y 481.629,Z 145.991,A -85,B 0,C 180,E1 -7073.376,E2 -7073.376} C_VEL
LIN {X 0,Y 481.678,Z 145.981,A -85,B 0,C 180,E1 -7076.328,E2 -7076.328} C_VEL
LIN {X 0,Y 481.652,Z 145.992,A -85,B 0,C 180,E1 -7079.418,E2 -7079.418} C_VEL
LIN {X 0,Y 481.702,Z 145.978,A -85,B 0,C 180,E1 -7082.168,E2 -7082.168} C_VEL
LIN {X 0,Y 481.72,Z 145.981,A -85,B 0,C 180,E1 -7084.97,E2 -7084.97} C_VEL
LIN {X 0,Y 481.681,Z 145.985,A -85,B 0,C 180,E1 -7087.966,E2 -7087.966} C_VEL
LIN {X 0,Y 481.512,Z 146.82,A -85,B 0,C 180,E1 -7088.376,E2 -7088.376} C_VEL
LIN {X 0,Y 480.824,Z 149.174,A -85,B 0,C 180,E1 -7088.854,E2 -7088.854} C_VEL
LIN {X 0,Y 476.099,Z 159.845,A -85,B 0,C 180,E1 -7090.777,E2 -7090.777} C_VEL
LIN {X 0,Y 475.766,Z 161.873,A -85,B 0,C 180,E1 -7091.18,E2 -7091.18} C_VEL
LIN {X 0,Y 475.427,Z 172.599,A -85,B 0,C 180,E1 -7093.282,E2 -7093.282} C_VEL
LIN {X 0,Y 478.203,Z 188.114,A -85,B 0,C 180,E1 -7093.637,E2 -7093.637} C_VEL
LIN {X 0,Y 477.513,Z 280.288,A -85,B 0,C 180,E1 -7095.047,E2 -7095.047} C_VEL
LIN {X 0,Y 477.179,Z 294.18,A -85,B 0,C 180,E1 -7095.446,E2 -7095.446} C_VEL
LIN {X 0,Y 476.816,Z 306.605,A -85,B 0,C 180,E1 -7095.979,E2 -7095.979} C_VEL
LIN {X 0,Y 476.439,Z 318.387,A -85,B 0,C 180,E1 -7096.669,E2 -7096.669} C_VEL
LIN {X 0,Y 476.043,Z 328.559,A -85,B 0,C 180,E1 -7097.423,E2 -7097.423} C_VEL
LIN {X 0,Y 475.535,Z 339.036,A -85,B 0,C 180,E1 -7098.383,E2 -7098.383} C_VEL
LIN {X 0,Y 475.131,Z 347.595,A -85,B 0,C 180,E1 -7099.345,E2 -7099.345} C_VEL
LIN {X 0,Y 474.743,Z 355.479,A -85,B 0,C 180,E1 -7100.413,E2 -7100.413} C_VEL
LIN {X 0,Y 474.381,Z 363.188,A -85,B 0,C 180,E1 -7101.695,E2 -7101.695} C_VEL
LIN {X 0,Y 474.103,Z 370.259,A -85,B 0,C 180,E1 -7103.189,E2 -7103.189} C_VEL
LIN {X 0,Y 473.976,Z 374.97,A -85,B 0,C 180,E1 -7104.469,E2 -7104.469} C_VEL
LIN {X 0,Y 473.847,Z 378.579,A -85,B 0,C 180,E1 -7105.747,E2 -7105.747} C_VEL
LIN {X 0,Y 473.861,Z 380.443,A -85,B 0,C 180,E1 -7106.599,E2 -7106.599} C_VEL
LIN {X 0,Y 473.772,Z 381.851,A -85,B 0,C 180,E1 -7107.449,E2 -7107.449} C_VEL
LIN {X 0,Y 473.691,Z 383.467,A -85,B 0,C 180,E1 -7109.15,E2 -7109.15} C_VEL
LIN {X 0,Y 473.672,Z 383.704,A -85,B 0,C 180,E1 -7110,E2 -7110} C_VEL
LIN {X 0,Y 473.69,Z 383.518,A -85,B 0,C 180,E1 -7110.85,E2 -7110.85} C_VEL
LIN {X 0,Y 473.773,Z 381.967,A -85,B 0,C 180,E1 -7112.551,E2 -7112.551} C_VEL
LIN {X 0,Y 473.86,Z 380.61,A -85,B 0,C 180,E1 -7113.401,E2 -7113.401} C_VEL
LIN {X 0,Y 473.814,Z 377.747,A -85,B 0,C 180,E1 -7114.679,E2 -7114.679} C_VEL
LIN {X 0,Y 474.044,Z 373.857,A -85,B 0,C 180,E1 -7115.957,E2 -7115.957} C_VEL
LIN {X 0,Y 474.146,Z 368.844,A -85,B 0,C 180,E1 -7117.238,E2 -7117.238} C_VEL
LIN {X 0,Y 474.425,Z 362.533,A -85,B 0,C 180,E1 -7118.519,E2 -7118.519} C_VEL
LIN {X 0,Y 474.77,Z 354.631,A -85,B 0,C 180,E1 -7119.801,E2 -7119.801} C_VEL
LIN {X 0,Y 475.247,Z 344.8,A -85,B 0,C 180,E1 -7121.084,E2 -7121.084} C_VEL
LIN {X 0,Y 475.815,Z 334.486,A -85,B 0,C 180,E1 -7122.15,E2 -7122.15} C_VEL
LIN {X 0,Y 476.216,Z 323.233,A -85,B 0,C 180,E1 -7123.086,E2 -7123.086} C_VEL
LIN {X 0,Y 476.66,Z 311.279,A -85,B 0,C 180,E1 -7123.862,E2 -7123.862} C_VEL
LIN {X 0,Y 477.124,Z 299.239,A -85,B 0,C 180,E1 -7124.447,E2 -7124.447} C_VEL
LIN {X 0,Y 477.396,Z 286.133,A -85,B 0,C 180,E1 -7124.902,E2 -7124.902} C_VEL
LIN {X 0,Y 477.627,Z 273.53,A -85,B 0,C 180,E1 -7125.167,E2 -7125.167} C_VEL
LIN {X 0,Y 478.138,Z 187.144,A -85,B 0,C 180,E1 -7126.472,E2 -7126.472} C_VEL
LIN {X 0,Y 475.405,Z 172.669,A -85,B 0,C 180,E1 -7126.799,E2 -7126.799} C_VEL
LIN {X 0,Y 475.922,Z 157.149,A -85,B 0,C 180,E1 -7129.855,E2 -7129.855} C_VEL
LIN {X 0,Y 475.707,Z 152.714,A -85,B 0,C 180,E1 -7130.767,E2 -7130.767} C_VEL
LIN {X 0,Y 474.639,Z 146.864,A -85,B 0,C 180,E1 -7132.069,E2 -7132.069} C_VEL
LIN {X 0,Y 474.673,Z 146.856,A -85,B 0,C 180,E1 -7135.428,E2 -7135.428} C_VEL
LIN {X 0,Y 474.647,Z 146.859,A -85,B 0,C 180,E1 -7138.282,E2 -7138.282} C_VEL
LIN {X 0,Y 474.599,Z 146.864,A -85,B 0,C 180,E1 -7141.217,E2 -7141.217} C_VEL
LIN {X 0,Y 474.621,Z 146.864,A -85,B 0,C 180,E1 -7144.242,E2 -7144.242} C_VEL
LIN {X 0,Y 474.591,Z 146.863,A -85,B 0,C 180,E1 -7147.383,E2 -7147.383} C_VEL
LIN {X 0,Y 474.618,Z 146.864,A -85,B 0,C 180,E1 -7150.657,E2 -7150.657} C_VEL
LIN {X 0,Y 474.602,Z 146.862,A -85,B 0,C 180,E1 -7153.481,E2 -7153.481} C_VEL
LIN {X 0,Y 474.602,Z 146.865,A -85,B 0,C 180,E1 -7156.519,E2 -7156.519} C_VEL
LIN {X 0,Y 474.617,Z 146.861,A -85,B 0,C 180,E1 -7159.342,E2 -7159.342} C_VEL
LIN {X 0,Y 474.61,Z 146.865,A -85,B 0,C 180,E1 -7161.704,E2 -7161.704} C_VEL
LIN {X 0,Y 474.624,Z 146.859,A -85,B 0,C 180,E1 -7164.725,E2 -7164.725} C_VEL
LIN {X 0,Y 474.635,Z 146.866,A -85,B 0,C 180,E1 -7167.788,E2 -7167.788} C_VEL
LIN {X 0,Y 474.623,Z 146.86,A -85,B 0,C 180,E1 -7170.884,E2 -7170.884} C_VEL
LIN {X 0,Y 474.661,Z 146.863,A -85,B 0,C 180,E1 -7173.628,E2 -7173.628} C_VEL
LIN {X 0,Y 474.635,Z 146.858,A -85,B 0,C 180,E1 -7176.641,E2 -7176.641} C_VEL
LIN {X 0,Y 474.656,Z 146.856,A -85,B 0,C 180,E1 -7180.09,E2 -7180.09} C_VEL
LIN {X 0,Y 474.65,Z 146.858,A -85,B 0,C 180,E1 -7182.774,E2 -7182.774} C_VEL
LIN {X 0,Y 474.648,Z 146.862,A -85,B 0,C 180,E1 -7185.421,E2 -7185.421} C_VEL
LIN {X 0,Y 474.704,Z 146.849,A -85,B 0,C 180,E1 -7188.037,E2 -7188.037} C_VEL
LIN {X 0,Y 474.727,Z 146.849,A -85,B 0,C 180,E1 -7191.486,E2 -7191.486} C_VEL
LIN {X 0,Y 474.77,Z 146.841,A -85,B 0,C 180,E1 -7194.052,E2 -7194.052} C_VEL
LIN {X 0,Y 474.894,Z 146.827,A -85,B 0,C 180,E1 -7197.455,E2 -7197.455} C_VEL
LIN {X 0,Y 474.911,Z 146.824,A -85,B 0,C 180,E1 -7200,E2 -7200} C_VEL
LIN {X 0,Y 474.893,Z 146.831,A -85,B 0,C 180,E1 -7202.545,E2 -7202.545} C_VEL
LIN {X 0,Y 474.77,Z 146.842,A -85,B 0,C 180,E1 -7205.948,E2 -7205.948} C_VEL
LIN {X 0,Y 474.726,Z 146.854,A -85,B 0,C 180,E1 -7208.514,E2 -7208.514} C_VEL
LIN {X 0,Y 474.703,Z 146.852,A -85,B 0,C 180,E1 -7211.962,E2 -7211.962} C_VEL
LIN {X 0,Y 474.699,Z 146.85,A -85,B 0,C 180,E1 -7215.456,E2 -7215.456} C_VEL
LIN {X 0,Y 474.662,Z 146.855,A -85,B 0,C 180,E1 -7219.01,E2 -7219.01} C_VEL
LIN {X 0,Y 474.587,Z 146.867,A -85,B 0,C 180,E1 -7221.729,E2 -7221.729} C_VEL
LIN {X 0,Y 474.638,Z 146.86,A -85,B 0,C 180,E1 -7224.494,E2 -7224.494} C_VEL
LIN {X 0,Y 474.679,Z 146.853,A -85,B 0,C 180,E1 -7227.334,E2 -7227.334} C_VEL
LIN {X 0,Y 474.603,Z 146.862,A -85,B 0,C 180,E1 -7230.81,E2 -7230.81} C_VEL
LIN {X 0,Y 474.636,Z 146.863,A -85,B 0,C 180,E1 -7233.984,E2 -7233.984} C_VEL
LIN {X 0,Y 474.565,Z 146.867,A -85,B 0,C 180,E1 -7236.898,E2 -7236.898} C_VEL
LIN {X 0,Y 474.608,Z 146.869,A -85,B 0,C 180,E1 -7239.645,E2 -7239.645} C_VEL
LIN {X 0,Y 474.6,Z 146.863,A -85,B 0,C 180,E1 -7242.234,E2 -7242.234} C_VEL
LIN {X 0,Y 474.616,Z 146.867,A -85,B 0,C 180,E1 -7245.298,E2 -7245.298} C_VEL
LIN {X 0,Y 474.608,Z 146.861,A -85,B 0,C 180,E1 -7248.214,E2 -7248.214} C_VEL
LIN {X 0,Y 474.609,Z 146.865,A -85,B 0,C 180,E1 -7251.543,E2 -7251.543} C_VEL
LIN {X 0,Y 474.623,Z 146.862,A -85,B 0,C 180,E1 -7254.726,E2 -7254.726} C_VEL
LIN {X 0,Y 474.634,Z 146.859,A -85,B 0,C 180,E1 -7257.788,E2 -7257.788} C_VEL
LIN {X 0,Y 474.599,Z 146.87,A -85,B 0,C 180,E1 -7260.891,E2 -7260.891} C_VEL
LIN {X 0,Y 474.593,Z 146.867,A -85,B 0,C 180,E1 -7263.625,E2 -7263.625} C_VEL
LIN {X 0,Y 474.659,Z 147.039,A -85,B 0,C 180,E1 -7264.872,E2 -7264.872} C_VEL
LIN {X 0,Y 476.668,Z 158.018,A -85,B 0,C 180,E1 -7267.001,E2 -7267.001} C_VEL
LIN {X 0,Y 475.999,Z 174.277,A -85,B 0,C 180,E1 -7269.923,E2 -7269.923} C_VEL
LIN {X 0,Y 475.321,Z 192.875,A -85,B 0,C 180,E1 -7273.221,E2 -7273.221} C_VEL
LIN {X 0,Y 478.049,Z 211,A -85,B 0,C 180,E1 -7273.614,E2 -7273.614} C_VEL
LIN {X 0,Y 477.423,Z 301.044,A -85,B 0,C 180,E1 -7274.99,E2 -7274.99} C_VEL
LIN {X 0,Y 477.071,Z 314.31,A -85,B 0,C 180,E1 -7275.36,E2 -7275.36} C_VEL
LIN {X 0,Y 476.68,Z 326.47,A -85,B 0,C 180,E1 -7275.866,E2 -7275.866} C_VEL
LIN {X 0,Y 476.16,Z 338.74,A -85,B 0,C 180,E1 -7276.558,E2 -7276.558} C_VEL
LIN {X 0,Y 475.731,Z 349.599,A -85,B 0,C 180,E1 -7277.353,E2 -7277.353} C_VEL
LIN {X 0,Y 475.247,Z 360.77,A -85,B 0,C 180,E1 -7278.376,E2 -7278.376} C_VEL
LIN {X 0,Y 474.815,Z 369.303,A -85,B 0,C 180,E1 -7279.338,E2 -7279.338} C_VEL
LIN {X 0,Y 474.47,Z 377.177,A -85,B 0,C 180,E1 -7280.408,E2 -7280.408} C_VEL
LIN {X 0,Y 474.158,Z 384.868,A -85,B 0,C 180,E1 -7281.691,E2 -7281.691} C_VEL
LIN {X 0,Y 473.927,Z 391.957,A -85,B 0,C 180,E1 -7283.187,E2 -7283.187} C_VEL
LIN {X 0,Y 473.847,Z 396.675,A -85,B 0,C 180,E1 -7284.468,E2 -7284.468} C_VEL
LIN {X 0,Y 473.733,Z 400.277,A -85,B 0,C 180,E1 -7285.746,E2 -7285.746} C_VEL
LIN {X 0,Y 473.764,Z 402.137,A -85,B 0,C 180,E1 -7286.598,E2 -7286.598} C_VEL
LIN {X 0,Y 473.741,Z 403.53,A -85,B 0,C 180,E1 -7287.449,E2 -7287.449} C_VEL
LIN {X 0,Y 473.689,Z 405.131,A -85,B 0,C 180,E1 -7289.15,E2 -7289.15} C_VEL
LIN {X 0,Y 473.671,Z 405.347,A -85,B 0,C 180,E1 -7290,E2 -7290} C_VEL
LIN {X 0,Y 473.689,Z 405.131,A -85,B 0,C 180,E1 -7290.85,E2 -7290.85} C_VEL
LIN {X 0,Y 473.741,Z 403.532,A -85,B 0,C 180,E1 -7292.551,E2 -7292.551} C_VEL
LIN {X 0,Y 473.765,Z 402.139,A -85,B 0,C 180,E1 -7293.402,E2 -7293.402} C_VEL
LIN {X 0,Y 473.761,Z 399.206,A -85,B 0,C 180,E1 -7294.68,E2 -7294.68} C_VEL
LIN {X 0,Y 473.831,Z 395.237,A -85,B 0,C 180,E1 -7295.96,E2 -7295.96} C_VEL
LIN {X 0,Y 474.018,Z 389.135,A -85,B 0,C 180,E1 -7297.454,E2 -7297.454} C_VEL
LIN {X 0,Y 474.275,Z 382.465,A -85,B 0,C 180,E1 -7298.736,E2 -7298.736} C_VEL
LIN {X 0,Y 474.613,Z 374.189,A -85,B 0,C 180,E1 -7300.02,E2 -7300.02} C_VEL
LIN {X 0,Y 475.012,Z 365.706,A -85,B 0,C 180,E1 -7301.089,E2 -7301.089} C_VEL
LIN {X 0,Y 475.551,Z 355.433,A -85,B 0,C 180,E1 -7302.138,E2 -7302.138} C_VEL
LIN {X 0,Y 475.894,Z 345.14,A -85,B 0,C 180,E1 -7302.993,E2 -7302.993} C_VEL
LIN {X 0,Y 476.399,Z 333.483,A -85,B 0,C 180,E1 -7303.762,E2 -7303.762} C_VEL
LIN {X 0,Y 476.837,Z 321.818,A -85,B 0,C 180,E1 -7304.347,E2 -7304.347} C_VEL
LIN {X 0,Y 477.246,Z 309.29,A -85,B 0,C 180,E1 -7304.798,E2 -7304.798} C_VEL
LIN {X 0,Y 477.477,Z 296.6,A -85,B 0,C 180,E1 -7305.09,E2 -7305.09} C_VEL
LIN {X 0,Y 478.007,Z 209.874,A -85,B 0,C 180,E1 -7306.403,E2 -7306.403} C_VEL
LIN {X 0,Y 475.287,Z 192.982,A -85,B 0,C 180,E1 -7306.759,E2 -7306.759} C_VEL
LIN {X 0,Y 475.887,Z 176.884,A -85,B 0,C 180,E1 -7309.609,E2 -7309.609} C_VEL
LIN {X 0,Y 476.52,Z 161.756,A -85,B 0,C 180,E1 -7312.32,E2 -7312.32} C_VEL
LIN {X 0,Y 476.534,Z 156.742,A -85,B 0,C 180,E1 -7313.236,E2 -7313.236} C_VEL
LIN {X 0,Y 474.63,Z 146.867,A -85,B 0,C 180,E1 -7315.186,E2 -7315.186} C_VEL
LIN {X 0,Y 474.605,Z 146.861,A -85,B 0,C 180,E1 -7318.285,E2 -7318.285} C_VEL
LIN {X 0,Y 474.594,Z 146.868,A -85,B 0,C 180,E1 -7321.218,E2 -7321.218} C_VEL
LIN {X 0,Y 474.62,Z 146.861,A -85,B 0,C 180,E1 -7324.242,E2 -7324.242} C_VEL
LIN {X 0,Y 474.589,Z 146.865,A -85,B 0,C 180,E1 -7327.384,E2 -7327.384} C_VEL
LIN {X 0,Y 474.604,Z 146.862,A -85,B 0,C 180,E1 -7329.644,E2 -7329.644} C_VEL
LIN {X 0,Y 474.581,Z 146.869,A -85,B 0,C 180,E1 -7332.938,E2 -7332.938} C_VEL
LIN {X 0,Y 474.603,Z 146.863,A -85,B 0,C 180,E1 -7335.894,E2 -7335.894} C_VEL
LIN {X 0,Y 474.622,Z 146.861,A -85,B 0,C 180,E1 -7339.041,E2 -7339.041} C_VEL
LIN {X 0,Y 474.608,Z 146.862,A -85,B 0,C 180,E1 -7341.704,E2 -7341.704} C_VEL
LIN {X 0,Y 474.622,Z 146.862,A -85,B 0,C 180,E1 -7344.725,E2 -7344.725} C_VEL
LIN {X 0,Y 474.635,Z 146.861,A -85,B 0,C 180,E1 -7347.788,E2 -7347.788} C_VEL
LIN {X 0,Y 474.606,Z 146.862,A -85,B 0,C 180,E1 -7350.888,E2 -7350.888} C_VEL
LIN {X 0,Y 474.616,Z 146.863,A -85,B 0,C 180,E1 -7353.626,E2 -7353.626} C_VEL
LIN {X 0,Y 474.634,Z 146.859,A -85,B 0,C 180,E1 -7356.642,E2 -7356.642} C_VEL
LIN {X 0,Y 474.654,Z 146.86,A -85,B 0,C 180,E1 -7360.089,E2 -7360.089} C_VEL
LIN {X 0,Y 474.637,Z 146.858,A -85,B 0,C 180,E1 -7362.774,E2 -7362.774} C_VEL
LIN {X 0,Y 474.648,Z 146.861,A -85,B 0,C 180,E1 -7365.421,E2 -7365.421} C_VEL
LIN {X 0,Y 474.704,Z 146.852,A -85,B 0,C 180,E1 -7368.038,E2 -7368.038} C_VEL
LIN {X 0,Y 474.726,Z 146.855,A -85,B 0,C 180,E1 -7371.486,E2 -7371.486} C_VEL
LIN {X 0,Y 474.771,Z 146.842,A -85,B 0,C 180,E1 -7374.052,E2 -7374.052} C_VEL
LIN {X 0,Y 474.894,Z 146.832,A -85,B 0,C 180,E1 -7377.455,E2 -7377.455} C_VEL
LIN {X 0,Y 474.911,Z 146.824,A -85,B 0,C 180,E1 -7380,E2 -7380} C_VEL
LIN {X 0,Y 474.894,Z 146.827,A -85,B 0,C 180,E1 -7382.545,E2 -7382.545} C_VEL
LIN {X 0,Y 474.761,Z 146.842,A -85,B 0,C 180,E1 -7385.948,E2 -7385.948} C_VEL
LIN {X 0,Y 474.726,Z 146.849,A -85,B 0,C 180,E1 -7388.514,E2 -7388.514} C_VEL
LIN {X 0,Y 474.704,Z 146.849,A -85,B 0,C 180,E1 -7391.963,E2 -7391.963} C_VEL
LIN {X 0,Y 474.7,Z 146.851,A -85,B 0,C 180,E1 -7395.456,E2 -7395.456} C_VEL
LIN {X 0,Y 474.666,Z 146.858,A -85,B 0,C 180,E1 -7399.01,E2 -7399.01} C_VEL
LIN {X 0,Y 474.588,Z 146.864,A -85,B 0,C 180,E1 -7401.729,E2 -7401.729} C_VEL
LIN {X 0,Y 474.657,Z 146.863,A -85,B 0,C 180,E1 -7404.493,E2 -7404.493} C_VEL
LIN {X 0,Y 474.681,Z 146.852,A -85,B 0,C 180,E1 -7407.335,E2 -7407.335} C_VEL
LIN {X 0,Y 474.606,Z 146.868,A -85,B 0,C 180,E1 -7410.23,E2 -7410.23} C_VEL
LIN {X 0,Y 474.643,Z 146.857,A -85,B 0,C 180,E1 -7413.22,E2 -7413.22} C_VEL
LIN {X 0,Y 474.589,Z 146.869,A -85,B 0,C 180,E1 -7416.324,E2 -7416.324} C_VEL
LIN {X 0,Y 474.628,Z 146.862,A -85,B 0,C 180,E1 -7419.648,E2 -7419.648} C_VEL
LIN {X 0,Y 474.616,Z 146.86,A -85,B 0,C 180,E1 -7422.934,E2 -7422.934} C_VEL
LIN {X 0,Y 474.611,Z 146.869,A -85,B 0,C 180,E1 -7425.895,E2 -7425.895} C_VEL
LIN {X 0,Y 474.629,Z 146.859,A -85,B 0,C 180,E1 -7429.041,E2 -7429.041} C_VEL
LIN {X 0,Y 474.611,Z 146.869,A -85,B 0,C 180,E1 -7431.704,E2 -7431.704} C_VEL
LIN {X 0,Y 474.624,Z 146.859,A -85,B 0,C 180,E1 -7434.726,E2 -7434.726} C_VEL
LIN {X 0,Y 474.636,Z 146.862,A -85,B 0,C 180,E1 -7437.788,E2 -7437.788} C_VEL
LIN {X 0,Y 474.625,Z 146.861,A -85,B 0,C 180,E1 -7440.885,E2 -7440.885} C_VEL
LIN {X 0,Y 474.663,Z 146.86,A -85,B 0,C 180,E1 -7443.629,E2 -7443.629} C_VEL
